               IF NOT "IX_MPO_RefSwitchOvenFeederOutside_I7" AND "IX_MPO_RefSwitchOvenFeederInside_I6"
                   AND "IX_MPO_RefSwitchVac_PosTurnTable_I5" AND NOT "IX_MPO_RefSwitchVac_PosOven_I8" THEN
                   "QX_MPO_M5_VacuumTowardsOven_Q7" := FALSE;
                   "QX_MPO_M5_VacuumTowardsTurnTable_Q8" := FALSE;
                   "QX_MPO_M4_OvenFeederRetract_Q5" := FALSE;
                   "QX_MPO_M4_OvenFeederExtend_Q6" := FALSE;
                   "QX_MPO_ValveOvenDoor_Q13" := FALSE;
                   #li_StepCase := 200;
               END_IF;

           200: // vacuum suction device down at turn table
               IF "IX_MPO_RefSwitchTurnTable_PosVac_I1" THEN
                   "QX_MPO_ValveLowering_Q12" := TRUE;

                   #lx_Start_TON_Wait := TRUE;
                   #lt_TON_Wait := T#2000ms;

                   IF #lfb_TON_Wait.Q THEN
                       #lx_Start_TON_Wait := FALSE;
                       #li_StepCase := 210;
                   END_IF;
               END_IF;

           210: // vacuum off
               "QX_MPO_ValveVacuum_Q11" := FALSE;

               #lx_Start_TON_Wait := TRUE;
               #lt_TON_Wait := T#2000ms;

               IF #lfb_TON_Wait.Q THEN
                   #lx_Start_TON_Wait := FALSE;
                   #li_StepCase := 220;
               END_IF;

           220: // vacuum suction device up
               "QX_MPO_ValveLowering_Q12" := FALSE;

               #lx_Start_TON_Wait := TRUE;
               #lt_TON_Wait := T#2000ms;

               IF #lfb_TON_Wait.Q THEN
                   #lx_Start_TON_Wait := FALSE;
                   IF "gtyp_MPO".Workpiece_Parameters.DoSaw THEN
                       #li_StepCase := 230;
                   ELSE    //Just skip the saw all together
                       #li_StepCase := 251;
                   END_IF;
               END_IF;

           230: // Position turn table saw
               IF NOT "IX_MPO_RefSwitchTurnTable_PosSaw_I4" AND NOT "IX_MPO_RefSwitchTurnTable_PosBelt_I2" AND "IX_MPO_RefSwitchTurnTable_PosVac_I1" THEN
                   "QX_MPO_M1_TurnTableClockwise_Q1" := TRUE;
                   "QX_MPO_M1_TurnTableCounterclockwise_Q2" := FALSE;
               ELSIF "IX_MPO_RefSwitchTurnTable_PosSaw_I4" OR "IX_MPO_RefSwitchTurnTable_PosBelt_I2" AND NOT "IX_MPO_RefSwitchTurnTable_PosVac_I1" THEN
                   "QX_MPO_M1_TurnTableClockwise_Q1" := FALSE;
                   "QX_MPO_M1_TurnTableCounterclockwise_Q2" := FALSE;

                   // Update workpiece state to saw on and update timestamp
                   "gtyp_MPO".Workpiece.Workpiece_States.x_atSaw := TRUE;
                   "gtyp_MPO".Workpiece.Workpiece_States.ldt_Saw := DT_TO_LDT(#ldt_MQTT);

                   #li_StepCase := 240;
               END_IF;

           240: // Start sawing
               "QX_MPO_M3_Saw_Q4" := TRUE;



               #lx_Start_TON_Wait := TRUE;
               #lt_TON_Wait := "gtyp_MPO".Workpiece_Parameters.SawTime; //Replaced the default sawing time of T#4000ms with the variable

               IF #lfb_TON_Wait.Q THEN
                   #li_Return_LDT := RD_SYS_T(#ldt_MQTT);
                   "gtyp_MPO".History[6].i_code := 600;
                   "gtyp_MPO".History[6].ldt_ts := DT_TO_LDT(#ldt_MQTT);

                   #lx_Start_TON_Wait := FALSE;

                   //TURN OFF SAW
                   "QX_MPO_M3_Saw_Q4" := FALSE;

                   // Update workpiece state to saw off and update timestamp
                   "gtyp_MPO".Workpiece.Workpiece_States.x_atSaw := FALSE;
                   "gtyp_MPO".Workpiece.Workpiece_States.ldt_Saw := DT_TO_LDT(#ldt_MQTT);

                   #li_StepCase := 250;
               END_IF;

           250: // Position turn table Pos Belt
               IF "IX_MPO_RefSwitchTurnTable_PosSaw_I4" AND NOT "IX_MPO_RefSwitchTurnTable_PosBelt_I2" AND NOT "IX_MPO_RefSwitchTurnTable_PosVac_I1" THEN
                   "QX_MPO_M1_TurnTableClockwise_Q1" := TRUE;
                   "QX_MPO_M1_TurnTableCounterclockwise_Q2" := FALSE;
               ELSIF NOT "IX_MPO_RefSwitchTurnTable_PosSaw_I4" AND "IX_MPO_RefSwitchTurnTable_PosBelt_I2" AND NOT "IX_MPO_RefSwitchTurnTable_PosVac_I1" THEN
                   "QX_MPO_M1_TurnTableClockwise_Q1" := FALSE;
                   "QX_MPO_M1_TurnTableCounterclockwise_Q2" := FALSE;
                   #li_StepCase := 260;
               END_IF;

           251: // Position turn table Pos Belt Directly (this has been added by me)
               IF NOT "IX_MPO_RefSwitchTurnTable_PosBelt_I2" THEN
                   "gtyp_MPO"."i_PWM_TurnTable" := 700;
                   "QX_MPO_M1_TurnTableClockwise_Q1" := TRUE;
                   "QX_MPO_M1_TurnTableCounterclockwise_Q2" := FALSE;
               ELSIF NOT "IX_MPO_RefSwitchTurnTable_PosSaw_I4" AND "IX_MPO_RefSwitchTurnTable_PosBelt_I2" AND NOT "IX_MPO_RefSwitchTurnTable_PosVac_I1" THEN
                   "gtyp_MPO"."i_PWM_TurnTable" := 1000;
                   "QX_MPO_M1_TurnTableClockwise_Q1" := FALSE;
                   "QX_MPO_M1_TurnTableCounterclockwise_Q2" := FALSE;
                   #li_StepCase := 260;
               END_IF;

           260: // put workpiece to belt
               "QX_MPO_ValveFeeder_Q14" := TRUE;

               #lx_Start_TON_Wait := TRUE;
               #lt_TON_Wait := T#1000ms;

               IF #lfb_TON_Wait.Q THEN
                   #lx_Start_TON_Wait := FALSE;
                   "QX_MPO_ValveFeeder_Q14" := FALSE;
                   "QX_MPO_Compressor_Q10" := FALSE;
                   #li_StepCase := 270;
               END_IF;

           270: // Position turn table Pos Vacuum
               IF "IX_MPO_RefSwitchTurnTable_PosSaw_I4" OR "IX_MPO_RefSwitchTurnTable_PosBelt_I2" OR NOT "IX_MPO_RefSwitchTurnTable_PosVac_I1" THEN
                   "QX_MPO_M1_TurnTableClockwise_Q1" := FALSE;
                   "QX_MPO_M1_TurnTableCounterclockwise_Q2" := TRUE;
               ELSIF NOT "IX_MPO_RefSwitchTurnTable_PosSaw_I4" AND NOT "IX_MPO_RefSwitchTurnTable_PosBelt_I2" AND "IX_MPO_RefSwitchTurnTable_PosVac_I1" THEN
                   "QX_MPO_M1_TurnTableClockwise_Q1" := FALSE;
                   "QX_MPO_M1_TurnTableCounterclockwise_Q2" := FALSE;
                   "QX_MPO_Compressor_Q10" := FALSE;
                   #li_StepCase := 280;
               END_IF;

           280: // Start conveyor belt
               "QX_MPO_M2_ConveyorBeltForward_Q3" := TRUE;

               #lx_Time_Error := TRUE;

               IF #lfb_TOF_ConveyerBelt_Out.Q THEN
                   "gtyp_SLD".History := "gtyp_MPO".History;
                   "gtyp_SLD".Workpiece := "gtyp_MPO".Workpiece;
                   "gtyp_MPO".Workpiece.s_id := '0';
                   "gtyp_MPO".Workpiece.s_state := '';
                   "gtyp_MPO".Workpiece.s_type := '';
                   FOR #ti_Counter := 1 TO 8 DO
                       "gtyp_MPO".History[#ti_Counter].i_code := 0;
                       "gtyp_MPO".History[#ti_Counter].ldt_ts := DT#1990-01-01-00:00:00;
                   END_FOR;

                   "gtyp_Interface_Dashboard".Subscribe.State_MPO.x_active := FALSE;

                   #lx_Time_Error := FALSE;
                   #li_StepCase := 290;
               END_IF;

               // runtime error
               IF #lfb_TON_Error.Q THEN
                   #li_Lights := 4;
                   #lx_Time_Error := FALSE;
                   "QX_MPO_M2_ConveyorBeltForward_Q3" := FALSE;
                   "gtyp_Interface_Dashboard".Subscribe.State_MPO.x_active := FALSE;
                   "gtyp_MPO".x_Error := TRUE;
                   "gtyp_MPO".s_ErrorMessage := 'MPO RUNTIME ERROR';
                   #li_StepCase := 0;
               END_IF;

           290: // wait for runtime on conveyor belt

               IF NOT #lfb_TOF_ConveyerBelt_Out.Q THEN
                   #lx_Start_TON_Wait := FALSE;
                   "QX_MPO_M2_ConveyorBeltForward_Q3" := FALSE;
                   #li_StepCase := 60;
               END_IF;
               // Statement section ELSE
           ELSE
               ;
       END_CASE;

       "QW_MPO_PWM_TurnTable_M1" := "gtyp_MPO"."i_PWM_TurnTable";
       "QW_MPO_PWM_Vacuum_M5" := "gtyp_MPO"."i_PWM_Vacuum";

   ELSE
       #li_Lights := 1;
       #lx_Init := TRUE;
       "gtyp_MPO".x_Start_Park_Position := FALSE;
       "gtyp_MPO".x_Park_Position_Reached := FALSE;
   END_IF;
END_FUNCTION_BLOCK

FUNCTION_BLOCK "PRG_MPO_Set_Park_Position"   // FB39, SCL
TITLE = Program Set Positioning HBW
{ S7_Optimized_Access := 'TRUE' }
AUTHOR : A.Schaefer
VERSION : 0.0
   VAR
      lx_Init : Bool;
      lx_Start_TON_Wait : Bool;
      lt_TON_Wait : Time;
      li_StepCase : Int;
      lfb_TON_Wait : TON_TIME;
      lfb_R_Trig_Start_Park_Pos : R_TRIG;
   END_VAR
BEGIN
   IF #lx_Init THEN

       // FB TON Wait
       #lfb_TON_Wait(IN := #lx_Start_TON_Wait,
                     PT := #lt_TON_Wait);

       #lfb_R_Trig_Start_Park_Pos(CLK := "gtyp_Setup".x_Park_Position
                                  OR "IX_Set_Park_Position");

       // Set Start Park Position   
       IF #lfb_R_Trig_Start_Park_Pos.Q THEN
           "gtyp_MPO".x_Start_Park_Position := TRUE;
           #li_StepCase := 0;
       END_IF;

       // not Start Park Pos Step 0
       IF NOT "gtyp_MPO".x_Start_Park_Position THEN
           #li_StepCase := 0;
       END_IF;

       // step chain HBW
       CASE #li_StepCase OF

           0:  // init
               #lx_Start_TON_Wait := FALSE;
               #li_StepCase := 10;

           10:  // Set Positioning activ?
               IF "gtyp_MPO".x_Start_Park_Position AND NOT "gtyp_MPO".x_Park_Position_Reached THEN
                   #li_StepCase := 20;
               END_IF;

           20: // Towards
               "QX_MPO_M5_VacuumTowardsTurnTable_Q8" := FALSE;
               "QX_MPO_M5_VacuumTowardsOven_Q7" := TRUE;
               #lx_Start_TON_Wait := TRUE;
               #lt_TON_Wait := T#4000ms;

               IF #lfb_TON_Wait.Q THEN
                   "QX_MPO_M5_VacuumTowardsTurnTable_Q8" := FALSE;
                   "QX_MPO_M5_VacuumTowardsOven_Q7" := FALSE;
                   #lx_Start_TON_Wait := FALSE;
                   #li_StepCase := 30;
               END_IF;

           30: // homing vertical axis
               "QX_MPO_M1_TurnTableClockwise_Q1" := TRUE;
               "QX_MPO_M1_TurnTableCounterclockwise_Q2" := FALSE;
               #lx_Start_TON_Wait := TRUE;
               #lt_TON_Wait := T#1000ms;

               IF #lfb_TON_Wait.Q THEN
                   "QX_MPO_M1_TurnTableClockwise_Q1" := FALSE;
                   "QX_MPO_M1_TurnTableCounterclockwise_Q2" := FALSE;
                   #lx_Start_TON_Wait := FALSE;
                   #li_StepCase := 40;
               END_IF;

           40: // Deciding which doing
               "gtyp_MPO".x_Park_Position_Reached := TRUE;


               // Statement section ELSE    
           ELSE
               ;
       END_CASE;

   ELSE
       #lx_Init := TRUE;
   END_IF;
END_FUNCTION_BLOCK

// folder: NFC

FUNCTION_BLOCK "PRG_NFC"   // FB8, SCL
TITLE = Program NFC
{ S7_Optimized_Access := 'TRUE' }
AUTHOR : A.Schaefer
VERSION : 0.0
   VAR
      lx_Init : Bool;
      lx_Start : Bool;
      lx_Time_Wait : Bool;
      lx_Time_Error : Bool;
      li_StepCase : Int;
      ldt_MQTT : Date_And_Time;
      ldt_Delete_old : LDT;
      ldt_Read_old : LDT;
      li_Return_LDT : Int;
      lfb_TON_Error : TON_TIME;
      lfb_TON_Wait : TON_TIME;
   END_VAR
BEGIN
   IF #lx_Init THEN

       // runtime monitoring error
       #lfb_TON_Error(IN := #lx_Time_Error,
                      PT := T#30s);

       // runtime monitoring read uid
       #lfb_TON_Wait(IN := #lx_Time_Wait,
                     PT := T#5s);

       // step chain NFC
       CASE #li_StepCase OF

           0:  // init
               #lx_Time_Wait := FALSE;
               "gtyp_VGR"."x_NFC_Completed" := FALSE;

               // delete and write first state to chip
               IF "gtyp_VGR".x_NFC_Start_First AND NOT "gtyp_VGR".x_Workpiece_NiO THEN
                   "gtyp_Interface_TXT_Controler".Subscribe.State_NFC_Device.Workpiece.s_state := '';
                   "gtyp_Interface_TXT_Controler".Subscribe.State_NFC_Device.Workpiece.s_type := '';

                   "gtyp_Interface_TXT_Controler".Publish.ActionButtonNFCModule.s_cmd := '';
                   #li_StepCase := 10;
                   // write color or processed finished to chip
               ELSIF "gtyp_VGR".x_NFC_Start AND NOT "gtyp_VGR".x_Workpiece_NiO THEN
                   "gtyp_Interface_TXT_Controler".Publish.ActionButtonNFCModule.s_cmd := '';
                   #li_StepCase := 40;
                   // read chip for delete HBW
               ELSIF "QX_SSC_LED_Green_Q5" AND NOT "gtyp_VGR".x_Workpiece_NiO THEN
                   #ldt_Read_old := "gtyp_Interface_Dashboard".Publish.ActionButtonNFCModule.ldt_ts;
                   "gtyp_VGR".x_NFC_Start_First := FALSE;
                   "gtyp_VGR".x_NFC_Start := FALSE;
                   "gtyp_Interface_TXT_Controler".Publish.ActionButtonNFCModule.s_cmd := '';
                   #li_StepCase := 60;
               END_IF;

           10: // delete

               "gtyp_Interface_TXT_Controler".Publish.ActionButtonNFCModule.s_cmd := 'delete';
               #li_Return_LDT := RD_SYS_T(#ldt_MQTT);
               "gtyp_Interface_TXT_Controler".Publish.ActionButtonNFCModule.ldt_ts := DT_TO_LDT(#ldt_MQTT);

               #li_StepCase := 20;

           20: // wait to answer from dashboard
               #lx_Time_Error := TRUE;
               IF ("gtyp_Interface_TXT_Controler".Subscribe.State_NFC_Device.ldt_ts > "gtyp_Interface_TXT_Controler".Publish.ActionButtonNFCModule.ldt_ts)
                   AND ("gtyp_Interface_TXT_Controler".Subscribe.State_NFC_Device.Workpiece.s_type = 'NONE')
                   AND ("gtyp_Interface_TXT_Controler".Subscribe.State_NFC_Device.Workpiece.s_state <> '')
                   AND ("gtyp_Interface_TXT_Controler".Subscribe.State_NFC_Device.Workpiece.s_id <> '') THEN
                   "gtyp_VGR".Workpiece.s_id := "gtyp_Interface_TXT_Controler".Subscribe.State_NFC_Device.Workpiece.s_id;
                   #lx_Time_Error := FALSE;
                   #li_StepCase := 30;
               END_IF;
               // runtime error
               IF #lfb_TON_Error.Q THEN
                   #lx_Time_Error := FALSE;
                   "gtyp_VGR".x_Workpiece_NiO := TRUE;
                   #li_StepCase := 0;
               END_IF;


           30: // wait of answer 
               IF "gtyp_Interface_TXT_Controler".Subscribe.State_NFC_Device.Workpiece.s_id <> '' THEN
                   #li_StepCase := 40;
               END_IF;

           40:  // write
               "gtyp_Interface_TXT_Controler".Publish.ActionButtonNFCModule.History := "gtyp_VGR".History;
               "gtyp_Interface_TXT_Controler".Publish.ActionButtonNFCModule.Workpiece.s_type := "gtyp_VGR".Workpiece.s_type;
               "gtyp_Interface_TXT_Controler".Publish.ActionButtonNFCModule.Workpiece.s_state := "gtyp_VGR".Workpiece.s_state;

               #li_Return_LDT := RD_SYS_T(#ldt_MQTT);

               "gtyp_Interface_TXT_Controler".Publish.ActionButtonNFCModule.s_cmd := 'write';
               "gtyp_Interface_TXT_Controler".Publish.ActionButtonNFCModule.ldt_ts := DT_TO_LDT(#ldt_MQTT);

               #li_StepCase := 50;

           50: // wait of answer write 
               #lx_Time_Error := TRUE;
               IF ("gtyp_Interface_TXT_Controler".Subscribe.State_NFC_Device.ldt_ts > "gtyp_Interface_TXT_Controler".Publish.ActionButtonNFCModule.ldt_ts) THEN
                   #lx_Time_Error := FALSE;
                   #li_StepCase := 80;
               END_IF;
               // runtime error
               IF #lfb_TON_Error.Q THEN
                   #lx_Time_Error := FALSE;
                   "gtyp_VGR".x_Workpiece_NiO := TRUE;
                   #li_StepCase := 0;
               END_IF;

           60: // read uid cmd

               #li_Return_LDT := RD_SYS_T(#ldt_MQTT);

               "gtyp_Interface_TXT_Controler".Publish.ActionButtonNFCModule.s_cmd := 'read_uid';
               "gtyp_Interface_TXT_Controler".Publish.ActionButtonNFCModule.ldt_ts := DT_TO_LDT(#ldt_MQTT);
               #lx_Time_Wait := TRUE;
               #li_StepCase := 70;

           70: // wait of answer read_uid 
               IF NOT "QX_SSC_LED_Green_Q5" OR #lfb_TON_Wait.Q OR ("gtyp_Interface_TXT_Controler".Subscribe.State_NFC_Device.ldt_ts > "gtyp_Interface_TXT_Controler".Publish.ActionButtonNFCModule.ldt_ts) THEN
                   IF LEN("gtyp_Interface_TXT_Controler".Subscribe.State_NFC_Device.Workpiece.s_id) = 8 THEN
                       "gtyp_Setup".x_Clean_Rack_HBW := TRUE;
                   END_IF;
                   #lx_Time_Wait := FALSE;
                   "gtyp_Interface_TXT_Controler".Subscribe.State_NFC_Device.Workpiece.s_id := '';
                   #li_StepCase := 0;
               END_IF;

           80: // completed

               "gtyp_VGR"."x_NFC_Completed" := TRUE;

               IF NOT "gtyp_VGR".x_NFC_Start AND NOT "gtyp_VGR".x_NFC_Start_First THEN
                   "gtyp_VGR"."x_NFC_Completed" := FALSE;
                   #lx_Start := FALSE;
                   #li_StepCase := 0;
               END_IF;

               // Statement section ELSE
           ELSE
               ;
       END_CASE;

   ELSE
       #lx_Init := TRUE;
   END_IF;
END_FUNCTION_BLOCK

// folder: Order

FUNCTION_BLOCK "PRG_Order"   // FB20, SCL
TITLE = Program Order
{ S7_Optimized_Access := 'TRUE' }
AUTHOR : A.Schaefer
VERSION : 0.0
   VAR
      lx_Init : Bool;
      li_StepCase : Int;
      lldt_ts_old : LDT;
      ldt_MQTT : Date_And_Time;
      li_Return_LDT : Int;
      lfb_TON_Wait : TON_TIME;
      lx_Start_TON_Wait : Bool;
   END_VAR
   VAR_TEMP
      ti_Que_Counter : Int;
      ti_Que_Output : Int;
   END_VAR
BEGIN
   IF #lx_Init THEN
       #lfb_TON_Wait(IN := #lx_Start_TON_Wait,
                     PT := T#20s);

       // step chain order
       CASE #li_StepCase OF

           0:  // init
               #lx_Start_TON_Wait := FALSE;
               #li_StepCase := 10;

           10: // check whether order button has been pressed (time stamp changes)

               IF ("gtyp_Interface_Dashboard".Publish.OrderWorkpieceButton.ldt_ts > #lldt_ts_old) THEN
                   #lldt_ts_old := "gtyp_Interface_Dashboard".Publish.OrderWorkpieceButton.ldt_ts;
                   IF ("Queue".i_Queue_Index < "Ci_Queue_Length") THEN
                       "Queue".Queue["Queue".i_Queue_Index] := "gtyp_Interface_Dashboard".Publish.OrderWorkpieceButton;
                       #li_Return_LDT := RD_SYS_T(#ldt_MQTT);
                       "gtyp_Interface_Dashboard".Subscribe.State_Order.ldt_ts := DT_TO_LDT(#ldt_MQTT);
                       "gtyp_Interface_Dashboard".Subscribe.State_Order.s_state := 'ORDERED';
                       "gtyp_Interface_Dashboard".Subscribe.State_Order.s_type := "Queue".Queue["Queue".i_Queue_Index].s_type;
                       "Queue".i_Queue_Index += 1;
                       IF ("Queue".i_Queue_Index = "Ci_Queue_Length") THEN
                           "Queue".x_Queue_Full := TRUE;
                       END_IF;
                   END_IF;
                   //Reset the parameters when the order has been processed
                   "gtyp_Interface_Dashboard".Publish.OrderWorkpieceButton.Workpiece_Parameters := "Queue".Queue["Ci_Queue_Length"].Workpiece_Parameters;
               END_IF;

               //There is an order in the que
               IF ("Queue".i_Queue_Index > 0) THEN
                   //The VGR is ready to start with the next product in the que
                   IF "gtyp_VGR".x_Ready_For_Order AND "gtyp_VGR".x_Ready_For_Outsource THEN
                       //We want to output the first order
                       FOR #ti_Que_Output := 0 TO "Queue".i_Queue_Index - 1 DO
                           IF ("Queue".Queue[#ti_Que_Output].s_type = 'RED' AND "gtyp_HBW".i_Red_Available = 0) THEN
                               CONTINUE;
                           ELSIF ("Queue".Queue[#ti_Que_Output].s_type = 'BLUE' AND "gtyp_HBW".i_Blue_Available = 0) THEN
                               CONTINUE;
                           ELSIF ("Queue".Queue[#ti_Que_Output].s_type = 'WHITE' AND "gtyp_HBW".i_White_Available = 0) THEN
                               CONTINUE;
                           END_IF;
                           //Possible order found
                           //Set index back
                           "Queue".i_Queue_Index -= 1;
                           "Queue".x_Queue_Full := FALSE;
                           //VGR is ready
                           "gtyp_VGR".x_Ready_For_Order := FALSE;
                           //Copy que to VGR
                           "gtyp_VGR".s_HBW_Outsource_Typ := "Queue".Queue[#ti_Que_Output].s_type;
                           "gtyp_VGR".Worpiece_Parameters := "Queue".Queue[#ti_Que_Output].Workpiece_Parameters;

                           //ADDED TO MAKE DISPLAYING PARAMETERS ON DASHBOARD EASIER
                           "gtyp_VGR".Workpiece.Workpiece_Parameters := "Queue".Queue[#ti_Que_Output].Workpiece_Parameters;
                           //Shift que
                           FOR #ti_Que_Counter := #ti_Que_Output TO "Ci_Queue_Length" - 1 DO
                               "Queue".Queue[#ti_Que_Counter] := "Queue".Queue[#ti_Que_Counter + 1];
                           END_FOR;
                           //Start the HBW and VGR
                           "gtyp_VGR".x_HBW_Outsource := TRUE;
                           EXIT;
                       END_FOR;
                   END_IF;
               END_IF;

               IF "gtyp_VGR".x_HBW_PickedUp THEN
                   "gtyp_VGR".x_HBW_Outsource := FALSE;
                   "gtyp_VGR".s_HBW_Outsource_Typ := '';
                   #li_StepCase := 0;
               END_IF;

               // Statement section ELSE
           ELSE
               ;
       END_CASE;

   ELSE
       #lx_Init := TRUE;
       "Queue".i_Queue_Index := 0;
       "Queue".x_Queue_Full := FALSE;
       #lldt_ts_old := LDT#1970-01-01-00:00:00;
   END_IF;
END_FUNCTION_BLOCK

// folder: SLD_Sorting_Line_With_Color_Detection

FUNCTION_BLOCK "PRG_SLD_Calibration_Color"   // FB33, SCL
TITLE = Program Calibration Color Sensor SLD
{ S7_Optimized_Access := 'TRUE' }
AUTHOR : A.Schaefer
VERSION : 0.0
   VAR
      lx_Init : Bool;
      lx_Start_TON_Wait : Bool;
      lx_Start_Positioning_m : Bool;
      lt_TON_Wait : Time;
      li_StepCase : Int;
      lw_ColorValueMin : Word;
      ldi_Pos_Horizontal : DInt;
      ldi_Pos_Vertical : DInt;
      lfb_R_Trig_Deaktivate : R_TRIG;
      lfb_TON_Wait : TON_TIME;
   END_VAR
BEGIN
   IF #lx_Init THEN

       // FB TON Wait
       #lfb_TON_Wait(IN := #lx_Start_TON_Wait,
                     PT := #lt_TON_Wait);

       #lfb_R_Trig_Deaktivate(CLK := NOT "gtyp_Setup".x_Color_Sensor_Calibration
                              OR NOT ("gtyp_Setup".i_Color_Sensor_Selection = 2));
       // Deaktivate step 0   
       IF #lfb_R_Trig_Deaktivate.Q THEN
           "gtyp_Setup".x_Calculate_Value_Color := FALSE;
           "gtyp_Setup".x_Set_Calib_Value_Color_Blue := FALSE;
           "gtyp_Setup".x_Set_Calib_Value_Color_Red := FALSE;
           "gtyp_Setup".x_Set_Calib_Value_Color_White := FALSE;
           "gtyp_Setup".w_Calib_ColorValue_Blue := 0;
           "gtyp_Setup".w_Calib_ColorValue_Red := 0;
           "gtyp_Setup".w_Calib_ColorValue_White := 0;
           "gtyp_Setup".w_Threshold_Red_Blue := 0;
           "gtyp_Setup".w_Threshold_White_Red := 0;
           "QX_SLD_M1_ConveyorBelt_Q1" := FALSE;
           #lw_ColorValueMin := 16#FF;
           #li_StepCase := 0;
       END_IF;

       // step chain HBW
       CASE #li_StepCase OF

           0:  // init
               #lx_Start_TON_Wait := FALSE;
               #li_StepCase := 10;

           10:  // Set Calibration activ?
               IF "gtyp_Setup".x_Color_Sensor_Calibration
                   AND ("gtyp_Setup".i_Color_Sensor_Selection = 2) THEN
                   "gtyp_Setup".x_Calculate_Value_Color := FALSE;
                   "gtyp_Setup".x_Set_Calib_Value_Color_Blue := FALSE;
                   "gtyp_Setup".x_Set_Calib_Value_Color_Red := FALSE;
                   "gtyp_Setup".x_Set_Calib_Value_Color_White := FALSE;
                   "gtyp_Setup".w_Calib_ColorValue_Blue := 0;
                   "gtyp_Setup".w_Calib_ColorValue_Red := 0;
                   "gtyp_Setup".w_Calib_ColorValue_White := 0;
                   "gtyp_Setup".w_Threshold_Red_Blue := 0;
                   "gtyp_Setup".w_Threshold_White_Red := 0;
                   "QX_SLD_M1_ConveyorBelt_Q1" := FALSE;
                   #lw_ColorValueMin := 16#FFFF;
                   #li_StepCase := 20;
               END_IF;

           20: // wait for set Values or Calculate

               IF NOT "IX_SLD_LightBarrierInlet_I2" THEN
                   "QX_SLD_M1_ConveyorBelt_Q1" := TRUE;
                   #lw_ColorValueMin := 16#FFFF;
               END_IF;

               IF #lw_ColorValueMin > "IW_SLD_ColorSensor_A4" THEN
                   #lw_ColorValueMin := "IW_SLD_ColorSensor_A4";
               END_IF;

               IF NOT "IX_SLD_LightBarrierBehindColorSensor_I3" THEN
                   "QX_SLD_M1_ConveyorBelt_Q1" := FALSE;
               END_IF;

               // Start new Positioning
               IF "gtyp_Setup".x_Set_Calib_Value_Color_Blue THEN
                   "gtyp_Setup".w_Calib_ColorValue_Blue := #lw_ColorValueMin;
                   "gtyp_Setup".x_Set_Calib_Value_Color_Blue := FALSE;
               ELSIF "gtyp_Setup".x_Set_Calib_Value_Color_Red THEN
                   "gtyp_Setup".w_Calib_ColorValue_Red := #lw_ColorValueMin;
                   "gtyp_Setup".x_Set_Calib_Value_Color_Red := FALSE;
               ELSIF "gtyp_Setup".x_Set_Calib_Value_Color_White THEN
                   "gtyp_Setup".w_Calib_ColorValue_White := #lw_ColorValueMin;
                   "gtyp_Setup".x_Set_Calib_Value_Color_White := FALSE;
               END_IF;

               "gtyp_Setup".w_Threshold_White_Red := "gtyp_Setup".w_Calib_ColorValue_White + (("gtyp_Setup".w_Calib_ColorValue_Red - "gtyp_Setup".w_Calib_ColorValue_White) / 2);
               "gtyp_Setup".w_Threshold_Red_Blue := "gtyp_Setup".w_Calib_ColorValue_Red + (("gtyp_Setup".w_Calib_ColorValue_Blue - "gtyp_Setup".w_Calib_ColorValue_Red) / 2);

               IF "gtyp_Setup".x_Calculate_Value_Color THEN
                   "gtyp_SLD".w_Threshold_White_Red := "gtyp_Setup".w_Threshold_White_Red;
                   "gtyp_SLD".w_Threshold_Red_Blue := "gtyp_Setup".w_Threshold_Red_Blue;
                   "gtyp_Setup".x_Calculate_Value_Color := FALSE;
               END_IF;

               // Statement section ELSE    
           ELSE
               ;
       END_CASE;

       IF ("gtyp_Setup".i_Color_Sensor_Selection = 2) THEN
           // Reload Pos Value
           "gtyp_Setup".w_Actual_ColorValue := "IW_SLD_ColorSensor_A4";
       END_IF;
   ELSE
       #lx_Init := TRUE;
   END_IF;
END_FUNCTION_BLOCK

FUNCTION_BLOCK "PRG_SLD_Set_Counter_Values"   // FB34, SCL
TITLE = Program Set counter Values SLD
{ S7_Optimized_Access := 'TRUE' }
AUTHOR : A.Schaefer
VERSION : 0.0
   VAR
      lx_Init : Bool;
      lfb_R_Trig_Calib_activ : R_TRIG;
   END_VAR
BEGIN
   IF #lx_Init THEN

       // Reload act. Counter Values
       IF NOT "gtyp_Setup".x_Counter_Value_Calibration THEN
           "gtyp_Setup".i_Calib_CounterValue_Blue := "gtyp_SLD".i_CounterValue_Blue;
           "gtyp_Setup".i_Calib_CounterValue_Red := "gtyp_SLD".i_CounterValue_Red;
           "gtyp_Setup".i_Calib_CounterValue_White := "gtyp_SLD".i_CounterValue_White;
       END_IF;

       // Set Counter Values   
       IF "gtyp_Setup".x_Set_CounterValues AND "gtyp_Setup".x_Counter_Value_Calibration THEN
           "gtyp_SLD".i_CounterValue_Blue := "gtyp_Setup".i_Calib_CounterValue_Blue;
           "gtyp_SLD".i_CounterValue_Red := "gtyp_Setup".i_Calib_CounterValue_Red;
           "gtyp_SLD".i_CounterValue_White := "gtyp_Setup".i_Calib_CounterValue_White;
           "gtyp_Setup".x_Set_CounterValues := FALSE;
       END_IF;

   ELSE
       #lx_Init := TRUE;
   END_IF;
END_FUNCTION_BLOCK

// folder: SSC_Sensor_Station_With_Camera

FUNCTION_BLOCK "PRG_SSC_Axis_Vertical"   // FB11, SCL
TITLE = Program Axis vertical SSC
{ S7_Optimized_Access := 'TRUE' }
AUTHOR : A.Schaefer
VERSION : 0.0
   VAR
      lx_Init : Bool;
      lfb_Vertical_Axis : "FB_Axis";
   END_VAR
BEGIN
   IF #lx_Init THEN

       // FB Axis vertical
       #lfb_Vertical_Axis(ini_Axis := 5,
                          indi_Increment := "gtyp_SSC".Vertical_Axis.di_Increment,
                          inx_Ref_Switch := "IX_SSC_RefSwitchVerticalAxis_I1",
                          inx_Referencing := "gtyp_SSC".Vertical_Axis.x_Reference,
                          inx_Start_Positioning := "gtyp_SSC".Vertical_Axis.x_Start_Positioning,
                          indi_Target_Position := "gtyp_SSC".Vertical_Axis.di_Target_Position,
                          ini_PWM := "gtyp_SSC".Vertical_Axis.i_PWM,
                          inouttyp_Config := "gtyp_SSC".Vertical_Axis.Config,
                          inouttyp_Setup := "gtyp_SetupAxis");

       "QX_SSC_M1_VerticalAxisUp_Q1" := #lfb_Vertical_Axis.outx_Motor_Pos;
       "QX_SSC_M1_VerticalAxisDown_Q2" := #lfb_Vertical_Axis.outx_Motor_Neg;
       "QW_SSC_PWM_Vertical_M1" := #lfb_Vertical_Axis.outi_Motor_PWM;
       "gtyp_SSC".Vertical_Axis.di_Actual_Position := #lfb_Vertical_Axis.outdi_Actual_Position;
       "gtyp_SSC".Vertical_Axis.x_Referenced := #lfb_Vertical_Axis.outx_Referenced;
       "gtyp_SSC".Vertical_Axis.x_Position_Reached := #lfb_Vertical_Axis.outx_Position_Reached;
   ELSE
       #lx_Init := TRUE;
   END_IF;
END_FUNCTION_BLOCK

FUNCTION_BLOCK "PRG_SSC_Ablauf"   // FB12, SCL
TITLE = Program Ablauf SSC
{ S7_Optimized_Access := 'TRUE' }
AUTHOR : A.Schaefer
VERSION : 0.0
   VAR
      lx_Init : Bool;
      lx_FirstCentre : Bool;
      lx_Start : Bool;
      lx_Start_TON_State : Bool;
      lt_TON_Wait : Time;
      li_StepCase : Int;
      ldi_TargetPosition_Horizontal : DInt;
      ldi_TargetPosition_Vertical : DInt;
      lldt_ts_old : LDT;
      ldt_write : Date_And_Time;
      li_Return_write : Int;
      ldt_MQTT : Date_And_Time;
      li_Return_LDT : Int;
      lx_Start_TON_Wait : Bool;
      ldi_StepHorizontal : DInt;
      ldi_StepVertical : DInt;
      lfb_TON_Wait : TON_TIME;
      lfb_TON_State : TON_TIME;
      lfb_F_TRIG_Set_Pos : F_TRIG;
   END_VAR
BEGIN
   IF #lx_Init THEN

       // Restart after set Positioning
       IF "gtyp_Setup".x_Set_Pos_Activ OR "gtyp_SSC".x_Start_Park_Position THEN
           #li_StepCase := 0;
       END_IF;

       // falling edge Set Pos
       #lfb_F_TRIG_Set_Pos(CLK := "gtyp_Setup".x_Set_Pos_Activ);

       IF #lfb_F_TRIG_Set_Pos.Q THEN
           #lx_FirstCentre := TRUE;
       END_IF;

       #lfb_TON_Wait(IN := #lx_Start_TON_Wait,
                     PT := #lt_TON_Wait);

       // wait time state
       #lfb_TON_State(IN := NOT #lx_Start_TON_State,
                      PT := T#2s);

       // state of the ssc cyclically transmitted to the cloud
       IF #lfb_TON_State.Q AND NOT #lx_Start_TON_State THEN
           #lx_Start_TON_State := TRUE;
           #li_Return_LDT := RD_SYS_T(#ldt_MQTT);
           "gtyp_Interface_Dashboard".Subscribe.PosPanTiltUnit.ldt_ts := DT_TO_LDT(#ldt_MQTT);
       END_IF;

       // restart wait time state
       IF NOT #lfb_TON_State.Q AND #lx_Start_TON_State THEN
           #lx_Start_TON_State := FALSE;
       END_IF;

       CASE #li_StepCase OF

           0:  // Init
               #lx_Start_TON_State := FALSE;
               "gtyp_SSC".Horizontal_Axis.x_Start_Positioning := FALSE;
               "gtyp_SSC".Vertical_Axis.x_Start_Positioning := FALSE;

               IF NOT "gtyp_Setup".x_Set_Pos_Activ AND NOT "gtyp_SSC".x_Start_Park_Position THEN
                   #li_StepCase := 10;
               END_IF;

           10: // Deciding which route to take 

               IF ("gtyp_Interface_Dashboard".Publish.PosPanTiltUnit.ldt_ts > #lldt_ts_old) OR #lx_FirstCentre THEN

                   #lldt_ts_old := "gtyp_Interface_Dashboard".Publish.PosPanTiltUnit.ldt_ts;

                   // convert the degrees to position
                   #ldi_StepHorizontal := REAL_TO_DINT("FC_Scale_linear"(inr_Y1 := DINT_TO_REAL("gtyp_SSC".Horizontal_Axis.Config.di_Neg_Soft_Switch),
                                                                                                             inr_Y2 := DINT_TO_REAL("gtyp_SSC".Horizontal_Axis.Config.di_Pos_Soft_Switch),
                                                                                                             inr_X1 := 0.0,
                                                                                                             inr_X2 := 180.0,
                                                                                                             inr_X := DINT_TO_REAL("gtyp_Interface_Dashboard".Publish.PosPanTiltUnit.i_degree)));
                   #ldi_StepVertical := REAL_TO_DINT("FC_Scale_linear"(inr_Y1 := DINT_TO_REAL("gtyp_SSC".Vertical_Axis.Config.di_Neg_Soft_Switch),
                                                                                                         inr_Y2 := DINT_TO_REAL("gtyp_SSC".Vertical_Axis.Config.di_Pos_Soft_Switch),
                                                                                                         inr_X1 := 0.0,
                                                                                                         inr_X2 := 180.0,
                                                                                                         inr_X := DINT_TO_REAL("gtyp_Interface_Dashboard".Publish.PosPanTiltUnit.i_degree)));
                   // Procedure - relmove_left
                   IF ("gtyp_Interface_Dashboard".Publish.PosPanTiltUnit.s_cmd = 'relmove_left')
                       AND (("gtyp_SSC".Horizontal_Axis.di_Actual_Position - #ldi_StepHorizontal) > "gtyp_SSC".Horizontal_Axis.Config.di_Neg_Soft_Switch + 15)
                       AND NOT "IX_SSC_RefSwitchHorizontalAxis_I2" THEN
                       #ldi_TargetPosition_Horizontal := "gtyp_SSC".Horizontal_Axis.di_Actual_Position - #ldi_StepHorizontal;
                       "gtyp_SSC".Horizontal_Axis.di_Target_Position := #ldi_TargetPosition_Horizontal;
                       "gtyp_SSC".Horizontal_Axis.x_Start_Positioning := TRUE;
                       #li_StepCase := 70;
                       // Procedure - relmove_right
                   ELSIF ("gtyp_Interface_Dashboard".Publish.PosPanTiltUnit.s_cmd = 'relmove_right')
                       AND (("gtyp_SSC".Horizontal_Axis.di_Actual_Position + #ldi_StepHorizontal) < "gtyp_SSC".Horizontal_Axis.Config.di_Pos_Soft_Switch - 15) THEN
                       #ldi_TargetPosition_Horizontal := "gtyp_SSC".Horizontal_Axis.di_Actual_Position + #ldi_StepHorizontal;
                       "gtyp_SSC".Horizontal_Axis.di_Target_Position := #ldi_TargetPosition_Horizontal;
                       "gtyp_SSC".Horizontal_Axis.x_Start_Positioning := TRUE;
                       #li_StepCase := 70;
                       // Procedure - relmove_up
                   ELSIF ("gtyp_Interface_Dashboard".Publish.PosPanTiltUnit.s_cmd = 'relmove_up')
                       AND (("gtyp_SSC".Vertical_Axis.di_Actual_Position + #ldi_StepHorizontal) < "gtyp_SSC".Vertical_Axis.Config.di_Pos_Soft_Switch - 15) THEN
                       #ldi_TargetPosition_Vertical := "gtyp_SSC".Vertical_Axis.di_Actual_Position + #ldi_StepVertical;
                       "gtyp_SSC".Vertical_Axis.di_Target_Position := #ldi_TargetPosition_Vertical;
                       "gtyp_SSC".Vertical_Axis.x_Start_Positioning := TRUE;
                       #li_StepCase := 80;
                       // Procedure - relmove_down
                   ELSIF ("gtyp_Interface_Dashboard".Publish.PosPanTiltUnit.s_cmd = 'relmove_down')
                       AND (("gtyp_SSC".Vertical_Axis.di_Actual_Position - #ldi_StepVertical) > "gtyp_SSC".Vertical_Axis.Config.di_Neg_Soft_Switch + 15)
                       AND NOT "IX_SSC_RefSwitchVerticalAxis_I1" THEN
                       #ldi_TargetPosition_Vertical := "gtyp_SSC".Vertical_Axis.di_Actual_Position - #ldi_StepVertical;
                       "gtyp_SSC".Vertical_Axis.di_Target_Position := #ldi_TargetPosition_Vertical;
                       "gtyp_SSC".Vertical_Axis.x_Start_Positioning := TRUE;
                       #li_StepCase := 80;
                       // Procedure - first 
                   ELSIF #lx_FirstCentre THEN
                       #li_StepCase := 20;
                       // Procedure - home
                   ELSIF ("gtyp_Interface_Dashboard".Publish.PosPanTiltUnit.s_cmd = 'home') THEN
                       #li_StepCase := 60;
                       // Procedure - start_pan
                   ELSIF ("gtyp_Interface_Dashboard".Publish.PosPanTiltUnit.s_cmd = 'start_pan')
                       AND ("gtyp_SSC".Horizontal_Axis.di_Actual_Position > "gtyp_SSC".Horizontal_Axis.Config.di_Neg_Soft_Switch + 15)
                       AND NOT "IX_SSC_RefSwitchHorizontalAxis_I2" THEN
                       #ldi_TargetPosition_Horizontal := "gtyp_SSC".Horizontal_Axis.Config.di_Neg_Soft_Switch + 15;
                       "gtyp_SSC".Horizontal_Axis.di_Target_Position := #ldi_TargetPosition_Horizontal;
                       "gtyp_SSC".Horizontal_Axis.x_Start_Positioning := TRUE;
                       #li_StepCase := 70;
                       // Procedure - end_pan
                   ELSIF ("gtyp_Interface_Dashboard".Publish.PosPanTiltUnit.s_cmd = 'end_pan')
                       AND ("gtyp_SSC".Horizontal_Axis.di_Actual_Position < "gtyp_SSC".Horizontal_Axis.Config.di_Pos_Soft_Switch - 15) THEN
                       #ldi_TargetPosition_Horizontal := "gtyp_SSC".Horizontal_Axis.Config.di_Pos_Soft_Switch - 15;
                       "gtyp_SSC".Horizontal_Axis.di_Target_Position := #ldi_TargetPosition_Horizontal;
                       "gtyp_SSC".Horizontal_Axis.x_Start_Positioning := TRUE;
                       #li_StepCase := 70;
                       // Procedure - start_tilt
                   ELSIF ("gtyp_Interface_Dashboard".Publish.PosPanTiltUnit.s_cmd = 'start_tilt')
                       AND ("gtyp_SSC".Vertical_Axis.di_Actual_Position > "gtyp_SSC".Vertical_Axis.Config.di_Neg_Soft_Switch + 15)
                       AND NOT "IX_SSC_RefSwitchVerticalAxis_I1" THEN
                       #ldi_TargetPosition_Vertical := "gtyp_SSC".Vertical_Axis.Config.di_Neg_Soft_Switch + 15;
                       "gtyp_SSC".Vertical_Axis.di_Target_Position := #ldi_TargetPosition_Vertical;
                       "gtyp_SSC".Vertical_Axis.x_Start_Positioning := TRUE;
                       #li_StepCase := 80;
                       // Procedure - end_tilt
                   ELSIF ("gtyp_Interface_Dashboard".Publish.PosPanTiltUnit.s_cmd = 'end_tilt')
                       AND ("gtyp_SSC".Vertical_Axis.di_Actual_Position < "gtyp_SSC".Vertical_Axis.Config.di_Pos_Soft_Switch - 15) THEN
                       #ldi_TargetPosition_Vertical := "gtyp_SSC".Vertical_Axis.Config.di_Pos_Soft_Switch - 15;
                       "gtyp_SSC".Vertical_Axis.di_Target_Position := #ldi_TargetPosition_Vertical;
                       "gtyp_SSC".Vertical_Axis.x_Start_Positioning := TRUE;
                       #li_StepCase := 80;
                   END_IF;
               END_IF;

           20: // homing vertical/horizontal axis
               "gtyp_SSC".Horizontal_Axis.x_Reference := TRUE;
               "gtyp_SSC".Vertical_Axis.x_Reference := TRUE;

               IF NOT "gtyp_SSC".Horizontal_Axis.x_Referenced AND NOT "gtyp_SSC".Vertical_Axis.x_Referenced THEN
                   #li_StepCase := 30;
               END_IF;

           30: // homed vertical/horizontal axis
               IF "gtyp_SSC".Horizontal_Axis.x_Referenced THEN
                   "gtyp_SSC".Horizontal_Axis.x_Reference := FALSE;
               END_IF;
               IF "gtyp_SSC".Vertical_Axis.x_Referenced THEN
                   "gtyp_SSC".Vertical_Axis.x_Reference := FALSE;
               END_IF;

               IF "gtyp_SSC".Horizontal_Axis.x_Referenced AND "gtyp_SSC".Vertical_Axis.x_Referenced THEN
                   "gtyp_SSC".Horizontal_Axis.x_Reference := FALSE;
                   "gtyp_SSC".Vertical_Axis.x_Reference := FALSE;
                   #lx_Start_TON_Wait := TRUE;
                   #li_StepCase := 40;
               END_IF;

           40: // wait sequence
               IF #lfb_TON_Wait.Q THEN
                   #lx_Start_TON_Wait := FALSE;
                   #li_StepCase := 50;
               END_IF;

           50: // Position horizontal/vertical axis and reached
               "gtyp_SSC".Horizontal_Axis.di_Target_Position := "gtyp_SSC".di_Pos_HBW_Horizontal;
               "gtyp_SSC".Horizontal_Axis.x_Start_Positioning := TRUE;
               "gtyp_SSC".Vertical_Axis.di_Target_Position := "gtyp_SSC".di_Pos_HBW_Vertical;
               "gtyp_SSC".Vertical_Axis.x_Start_Positioning := TRUE;

               IF ("gtyp_SSC".Horizontal_Axis.di_Actual_Position <= ("gtyp_SSC".di_Pos_HBW_Horizontal + "gtyp_SSC".Horizontal_Axis.Config.di_Pos_Window))
                   AND ("gtyp_SSC".Horizontal_Axis.di_Actual_Position >= ("gtyp_SSC".di_Pos_HBW_Horizontal - "gtyp_SSC".Horizontal_Axis.Config.di_Pos_Window))
                   AND "gtyp_SSC".Horizontal_Axis.x_Position_Reached THEN
                   "gtyp_SSC".Horizontal_Axis.x_Start_Positioning := FALSE;
               END_IF;

               IF ("gtyp_SSC".Vertical_Axis.di_Actual_Position <= ("gtyp_SSC".di_Pos_HBW_Vertical + "gtyp_SSC".Vertical_Axis.Config.di_Pos_Window))
                   AND ("gtyp_SSC".Vertical_Axis.di_Actual_Position >= ("gtyp_SSC".di_Pos_HBW_Vertical - "gtyp_SSC".Vertical_Axis.Config.di_Pos_Window))
                   AND "gtyp_SSC".Vertical_Axis.x_Position_Reached THEN
                   "gtyp_SSC".Vertical_Axis.x_Start_Positioning := FALSE;
               END_IF;

               IF ("gtyp_SSC".Horizontal_Axis.di_Actual_Position <= ("gtyp_SSC".di_Pos_HBW_Horizontal + "gtyp_SSC".Horizontal_Axis.Config.di_Pos_Window))
                   AND ("gtyp_SSC".Horizontal_Axis.di_Actual_Position >= ("gtyp_SSC".di_Pos_HBW_Horizontal - "gtyp_SSC".Horizontal_Axis.Config.di_Pos_Window))
                   AND "gtyp_SSC".Horizontal_Axis.x_Position_Reached
                   AND ("gtyp_SSC".Vertical_Axis.di_Actual_Position <= ("gtyp_SSC".di_Pos_HBW_Vertical + "gtyp_SSC".Vertical_Axis.Config.di_Pos_Window))
                   AND ("gtyp_SSC".Vertical_Axis.di_Actual_Position >= ("gtyp_SSC".di_Pos_HBW_Vertical - "gtyp_SSC".Vertical_Axis.Config.di_Pos_Window))
                   AND "gtyp_SSC".Vertical_Axis.x_Position_Reached THEN
                   "gtyp_SSC".Horizontal_Axis.x_Start_Positioning := FALSE;
                   "gtyp_SSC".Vertical_Axis.x_Start_Positioning := FALSE;
                   #lx_FirstCentre := FALSE;
                   #li_StepCase := 90;
               END_IF;

           60: // Position Centre horizontal/vertical axis and reached
               "gtyp_SSC".Horizontal_Axis.di_Target_Position := "gtyp_SSC".di_Pos_Centre_Horizontal;
               "gtyp_SSC".Horizontal_Axis.x_Start_Positioning := TRUE;
               "gtyp_SSC".Vertical_Axis.di_Target_Position := "gtyp_SSC".di_Pos_Centre_Vertical;
               "gtyp_SSC".Vertical_Axis.x_Start_Positioning := TRUE;

               IF ("gtyp_SSC".Horizontal_Axis.di_Actual_Position <= ("gtyp_SSC".di_Pos_Centre_Horizontal + "gtyp_SSC".Horizontal_Axis.Config.di_Pos_Window))
                   AND ("gtyp_SSC".Horizontal_Axis.di_Actual_Position >= ("gtyp_SSC".di_Pos_Centre_Horizontal - "gtyp_SSC".Horizontal_Axis.Config.di_Pos_Window))
                   AND "gtyp_SSC".Horizontal_Axis.x_Position_Reached THEN
                   "gtyp_SSC".Horizontal_Axis.x_Start_Positioning := FALSE;
               END_IF;

               IF ("gtyp_SSC".Vertical_Axis.di_Actual_Position <= ("gtyp_SSC".di_Pos_Centre_Vertical + "gtyp_SSC".Vertical_Axis.Config.di_Pos_Window))
                   AND ("gtyp_SSC".Vertical_Axis.di_Actual_Position >= ("gtyp_SSC".di_Pos_Centre_Vertical - "gtyp_SSC".Vertical_Axis.Config.di_Pos_Window))
                   AND "gtyp_SSC".Vertical_Axis.x_Position_Reached THEN
                   "gtyp_SSC".Vertical_Axis.x_Start_Positioning := FALSE;
               END_IF;

               IF ("gtyp_SSC".Horizontal_Axis.di_Actual_Position <= ("gtyp_SSC".di_Pos_Centre_Horizontal + "gtyp_SSC".Horizontal_Axis.Config.di_Pos_Window))
                   AND ("gtyp_SSC".Horizontal_Axis.di_Actual_Position >= ("gtyp_SSC".di_Pos_Centre_Horizontal - "gtyp_SSC".Horizontal_Axis.Config.di_Pos_Window))
                   AND "gtyp_SSC".Horizontal_Axis.x_Position_Reached
                   AND ("gtyp_SSC".Vertical_Axis.di_Actual_Position <= ("gtyp_SSC".di_Pos_Centre_Vertical + "gtyp_SSC".Vertical_Axis.Config.di_Pos_Window))
                   AND ("gtyp_SSC".Vertical_Axis.di_Actual_Position >= ("gtyp_SSC".di_Pos_Centre_Vertical - "gtyp_SSC".Vertical_Axis.Config.di_Pos_Window))
                   AND "gtyp_SSC".Vertical_Axis.x_Position_Reached THEN
                   "gtyp_SSC".Horizontal_Axis.x_Start_Positioning := FALSE;
                   "gtyp_SSC".Vertical_Axis.x_Start_Positioning := FALSE;
                   #lx_FirstCentre := FALSE;
                   #li_StepCase := 90;
               END_IF;

           70: // Position horizontal axis reached
               IF ("gtyp_SSC".Horizontal_Axis.di_Actual_Position <= (#ldi_TargetPosition_Horizontal + "gtyp_SSC".Horizontal_Axis.Config.di_Pos_Window))
                   AND ("gtyp_SSC".Horizontal_Axis.di_Actual_Position >= (#ldi_TargetPosition_Horizontal - "gtyp_SSC".Horizontal_Axis.Config.di_Pos_Window))
                   AND "gtyp_SSC".Horizontal_Axis.x_Position_Reached THEN
                   "gtyp_SSC".Horizontal_Axis.x_Start_Positioning := FALSE;
                   #li_StepCase := 90;
               END_IF;

           80: // Position vertical axis reached
               IF ("gtyp_SSC".Vertical_Axis.di_Actual_Position <= (#ldi_TargetPosition_Vertical + "gtyp_SSC".Vertical_Axis.Config.di_Pos_Window))
                   AND ("gtyp_SSC".Vertical_Axis.di_Actual_Position >= (#ldi_TargetPosition_Vertical - "gtyp_SSC".Vertical_Axis.Config.di_Pos_Window))
                   AND "gtyp_SSC".Vertical_Axis.x_Position_Reached THEN
                   "gtyp_SSC".Vertical_Axis.x_Start_Positioning := FALSE;
                   #li_StepCase := 90;
               END_IF;

           90: // convert the position to degrees
               "gtyp_Interface_Dashboard".Subscribe.PosPanTiltUnit.r_pan := "FC_Scale_linear"(inr_Y1 := -1.0,
                                                                                              inr_Y2 := 1.0,
                                                                                              inr_X1 := DINT_TO_REAL("gtyp_SSC".Horizontal_Axis.Config.di_Neg_Soft_Switch),
                                                                                              inr_X2 := DINT_TO_REAL("gtyp_SSC".Horizontal_Axis.Config.di_Pos_Soft_Switch),
                                                                                              inr_X := "gtyp_SSC".Horizontal_Axis.di_Actual_Position);
               "gtyp_Interface_Dashboard".Subscribe.PosPanTiltUnit.r_tilt := "FC_Scale_linear"(inr_Y1 := -1.0,
                                                                                               inr_Y2 := 1.0,
                                                                                               inr_X1 := DINT_TO_REAL("gtyp_SSC".Vertical_Axis.Config.di_Neg_Soft_Switch),
                                                                                               inr_X2 := DINT_TO_REAL("gtyp_SSC".Vertical_Axis.Config.di_Pos_Soft_Switch),
                                                                                               inr_X := "gtyp_SSC".Vertical_Axis.di_Actual_Position);

               #li_Return_write := RD_SYS_T(#ldt_write);
               "gtyp_Interface_Dashboard".Subscribe.PosPanTiltUnit.ldt_ts := DT_TO_LDT(#ldt_write);
               #lx_Start_TON_Wait := TRUE;
               #li_StepCase := 100;

           100:// wait sequence
               IF #lfb_TON_Wait.Q THEN
                   #lx_Start_TON_Wait := FALSE;
                   #li_StepCase := 0;
               END_IF;
               // Statement section ELSE        
           ELSE
               ;
       END_CASE;

   ELSE
       #lx_Init := TRUE;
       #lx_FirstCentre := TRUE;

       "gtyp_SSC".x_Start_Park_Position := FALSE;
       "gtyp_SSC".x_Park_Position_Reached := FALSE;
       "gtyp_SSC".x_Error := FALSE;
   END_IF;
END_FUNCTION_BLOCK

FUNCTION_BLOCK "PRG_SSC_Set_Positioning"   // FB13, SCL
TITLE = Program Set Positioning SSC
{ S7_Optimized_Access := 'TRUE' }
AUTHOR : A.Schaefer
VERSION : 0.0
   VAR
      lx_Init : Bool;
      lx_Start_TON_Wait : Bool;
      lx_Start_Positioning_m : Bool;
      lt_TON_Wait : Time;
      li_StepCase : Int;
      ldi_Pos_Horizontal : DInt;
      ldi_Pos_Vertical : DInt;
      lfb_R_Trig_Deaktivate : R_TRIG;
      lfb_TON_Wait : TON_TIME;
   END_VAR
BEGIN
   IF #lx_Init THEN

       // FB TON Wait
       #lfb_TON_Wait(IN := #lx_Start_TON_Wait,
                     PT := #lt_TON_Wait);

       #lfb_R_Trig_Deaktivate(CLK := NOT "gtyp_Setup".x_Set_Pos_Activ
                              OR NOT (("gtyp_Setup".i_Pos_Selection > 0)
                              AND ("gtyp_Setup".i_Pos_Selection < 21)));
       // Deaktivate step 10   
       IF #lfb_R_Trig_Deaktivate.Q THEN
           "gtyp_SSC".Horizontal_Axis.x_Start_Positioning := FALSE;
           "gtyp_SSC".Vertical_Axis.x_Start_Positioning := FALSE;
           "gtyp_SSC".Horizontal_Axis.x_Reference := FALSE;
           "gtyp_SSC".Vertical_Axis.x_Reference := FALSE;
           "gtyp_Setup".x_Start_Positioning := FALSE;
           "gtyp_Setup".x_Final_Positioning := FALSE;
           "gtyp_Setup".x_Home_Positioning := FALSE;
           "gtyp_Setup".x_Start_Offset := FALSE;
           #lx_Start_Positioning_m := FALSE;
           IF (#li_StepCase > 10) THEN
               #li_StepCase := 70;
           END_IF;
       END_IF;

       // Set Positioning activ?
       IF "gtyp_Setup".x_Set_Pos_Activ
           AND (("gtyp_Setup".i_Pos_Selection > 0)
           AND ("gtyp_Setup".i_Pos_Selection < 21))
           AND ((#li_StepCase = 40)
           OR (#li_StepCase = 60)) THEN

           // Deciding which Position
           // Position - Centre
           IF "gtyp_Setup".i_Pos_Selection = 1 THEN
               #ldi_Pos_Horizontal := "gtyp_SSC".di_Pos_Centre_Horizontal;
               #ldi_Pos_Vertical := "gtyp_SSC".di_Pos_Centre_Vertical;
               // Position - HBW 
           ELSIF "gtyp_Setup".i_Pos_Selection = 2 THEN
               #ldi_Pos_Horizontal := "gtyp_SSC".di_Pos_HBW_Horizontal;
               #ldi_Pos_Vertical := "gtyp_SSC".di_Pos_HBW_Vertical;
           END_IF;
       END_IF;

       // Set Positioning activ?
       IF NOT "gtyp_Setup".x_Set_Pos_Activ THEN
           "gtyp_Setup".i_Pos_Selection := 0;
       END_IF;

       // step chain HBW
       CASE #li_StepCase OF

           0:  // init
               #lx_Start_TON_Wait := FALSE;
               #li_StepCase := 10;

           10:  // Set Positioning activ?
               IF "gtyp_Setup".x_Set_Pos_Activ
                   AND (("gtyp_Setup".i_Pos_Selection > 0)
                   AND ("gtyp_Setup".i_Pos_Selection < 21)) THEN
                   "gtyp_SSC".Horizontal_Axis.x_Start_Positioning := FALSE;
                   "gtyp_SSC".Vertical_Axis.x_Start_Positioning := FALSE;
                   "gtyp_SSC".Horizontal_Axis.x_Reference := FALSE;
                   "gtyp_SSC".Vertical_Axis.x_Reference := FALSE;
                   "gtyp_Setup".x_Start_Positioning := FALSE;
                   "gtyp_Setup".x_Final_Positioning := FALSE;
                   "gtyp_Setup".x_Home_Positioning := FALSE;
                   "gtyp_Setup".x_Start_Offset := FALSE;
                   #li_StepCase := 20;
               END_IF;

           20: //homing vertical/horizontal axis

               "gtyp_SSC".Horizontal_Axis.x_Reference := TRUE;
               "gtyp_SSC".Vertical_Axis.x_Reference := TRUE;

               IF NOT "gtyp_SSC".Horizontal_Axis.x_Referenced AND NOT "gtyp_SSC".Vertical_Axis.x_Referenced THEN
                   #li_StepCase := 30;
               END_IF;

           30: // homed vertical/horizontal axis
               IF "gtyp_SSC".Horizontal_Axis.x_Referenced THEN
                   "gtyp_SSC".Horizontal_Axis.x_Reference := FALSE;
               END_IF;
               IF "gtyp_SSC".Vertical_Axis.x_Referenced THEN
                   "gtyp_SSC".Vertical_Axis.x_Reference := FALSE;
               END_IF;

               IF "gtyp_SSC".Horizontal_Axis.x_Referenced AND "gtyp_SSC".Vertical_Axis.x_Referenced THEN
                   "gtyp_SSC".Horizontal_Axis.x_Reference := FALSE;
                   "gtyp_SSC".Vertical_Axis.x_Reference := FALSE;
                   #li_StepCase := 40;
               END_IF;

           40:  // Start Positioning Step next
               IF "gtyp_Setup".x_Start_Positioning OR #lx_Start_Positioning_m THEN
                   #lx_Start_Positioning_m := FALSE;
                   #li_StepCase := 50;
               END_IF;

           50: // Position vertical/horizontal HBW
               "gtyp_SSC".Horizontal_Axis.di_Target_Position := #ldi_Pos_Horizontal;
               "gtyp_SSC".Horizontal_Axis.x_Start_Positioning := TRUE;
               "gtyp_SSC".Vertical_Axis.di_Target_Position := #ldi_Pos_Vertical;
               "gtyp_SSC".Vertical_Axis.x_Start_Positioning := TRUE;

               IF ("gtyp_SSC".Horizontal_Axis.di_Actual_Position <= (#ldi_Pos_Horizontal + "gtyp_SSC".Horizontal_Axis.Config.di_Pos_Window))
                   AND ("gtyp_SSC".Horizontal_Axis.di_Actual_Position >= (#ldi_Pos_Horizontal - "gtyp_SSC".Horizontal_Axis.Config.di_Pos_Window))
                   AND "gtyp_SSC".Horizontal_Axis.x_Position_Reached THEN
                   "gtyp_SSC".Horizontal_Axis.x_Start_Positioning := FALSE;
               END_IF;

               IF ("gtyp_SSC".Vertical_Axis.di_Actual_Position <= (#ldi_Pos_Vertical + "gtyp_SSC".Vertical_Axis.Config.di_Pos_Window))
                   AND ("gtyp_SSC".Vertical_Axis.di_Actual_Position >= (#ldi_Pos_Vertical - "gtyp_SSC".Vertical_Axis.Config.di_Pos_Window))
                   AND "gtyp_SSC".Vertical_Axis.x_Position_Reached THEN
                   "gtyp_SSC".Vertical_Axis.x_Start_Positioning := FALSE;
               END_IF;

               IF ("gtyp_SSC".Horizontal_Axis.di_Actual_Position <= (#ldi_Pos_Horizontal + "gtyp_SSC".Horizontal_Axis.Config.di_Pos_Window))
                   AND ("gtyp_SSC".Horizontal_Axis.di_Actual_Position >= (#ldi_Pos_Horizontal - "gtyp_SSC".Horizontal_Axis.Config.di_Pos_Window))
                   AND "gtyp_SSC".Horizontal_Axis.x_Position_Reached
                   AND ("gtyp_SSC".Vertical_Axis.di_Actual_Position <= (#ldi_Pos_Vertical + "gtyp_SSC".Vertical_Axis.Config.di_Pos_Window))
                   AND ("gtyp_SSC".Vertical_Axis.di_Actual_Position >= (#ldi_Pos_Vertical - "gtyp_SSC".Vertical_Axis.Config.di_Pos_Window))
                   AND "gtyp_SSC".Vertical_Axis.x_Position_Reached THEN
                   "gtyp_SSC".Horizontal_Axis.x_Start_Positioning := FALSE;
                   "gtyp_SSC".Vertical_Axis.x_Start_Positioning := FALSE;
                   "gtyp_Setup".x_Start_Positioning := FALSE;
                   #li_StepCase := 60;
               END_IF;

           60: // Deciding which doing

               // Start new Positioning
               IF "gtyp_Setup".x_Start_Positioning OR "gtyp_Setup".x_Home_Positioning THEN
                   #lx_Start_Positioning_m := TRUE;
                   #li_StepCase := 10;
               ELSIF #lfb_R_Trig_Deaktivate.Q THEN
                   "gtyp_Setup".x_Home_Positioning := FALSE;
                   #li_StepCase := 70;
               END_IF;

           70: //homing vertical/horizontal axis

               "gtyp_SSC".Horizontal_Axis.x_Reference := TRUE;
               "gtyp_SSC".Vertical_Axis.x_Reference := TRUE;

               IF NOT "gtyp_SSC".Horizontal_Axis.x_Referenced AND NOT "gtyp_SSC".Vertical_Axis.x_Referenced THEN
                   #li_StepCase := 80;
               END_IF;

           80: // homed vertical/horizontal axis
               IF "gtyp_SSC".Horizontal_Axis.x_Referenced THEN
                   "gtyp_SSC".Horizontal_Axis.x_Reference := FALSE;
               END_IF;
               IF "gtyp_SSC".Vertical_Axis.x_Referenced THEN
                   "gtyp_SSC".Vertical_Axis.x_Reference := FALSE;
               END_IF;

               IF "gtyp_SSC".Horizontal_Axis.x_Referenced AND "gtyp_SSC".Vertical_Axis.x_Referenced THEN
                   "gtyp_SSC".Horizontal_Axis.x_Reference := FALSE;
                   "gtyp_SSC".Vertical_Axis.x_Reference := FALSE;
                   #li_StepCase := 0;
               END_IF;

               // Statement section ELSE    
           ELSE
               ;
       END_CASE;

       IF (("gtyp_Setup".i_Pos_Selection > 0)
           AND ("gtyp_Setup".i_Pos_Selection < 21)) THEN
           // Reload Pos Value
           "gtyp_Setup".di_Pos_Horizontal := #ldi_Pos_Horizontal;
           "gtyp_Setup".di_Pos_Vertical := #ldi_Pos_Vertical;
           "gtyp_Setup".di_Pos_Rotate := 0;
       END_IF;
   ELSE
       #lx_Init := TRUE;
   END_IF;
END_FUNCTION_BLOCK

FUNCTION_BLOCK "PRG_SSC_Light"   // FB21, SCL
TITLE = Program Lights
{ S7_Optimized_Access := 'TRUE' }
AUTHOR : A.Schaefer
VERSION : 0.0
   VAR
      lx_Init : Bool;
      lx_Start : Bool;
      li_StepCase : Int;
      ldt_MQTT : Date_And_Time;
      lldt_ts_old : LDT;
      li_Return_LDT : Int;
      lfb_TOF_Camera : TOF_TIME;
      lfb_TON_Schritt : TON_TIME;
      lfb_blinker_cam : "FB_Blinker";
      lfb_blinker_config : "FB_Blinker";
      lx_StartTimer : Bool;
   END_VAR
BEGIN
   IF #lx_Init THEN

       // if camera sen picture - Red light flash
       IF "gtyp_Interface_Dashboard".Subscribe.CameraPicture.ldt_ts > #lldt_ts_old THEN
           #lldt_ts_old := "gtyp_Interface_Dashboard".Subscribe.CameraPicture.ldt_ts;
           #lfb_blinker_cam(int_periodendauer := T#50ms);
       END_IF;

       // reload flash
       "QX_SSC_LED_Red_Online_Q8" := #lfb_blinker_cam.outx_blinker;

       // FB flash config
       #lfb_blinker_config(int_periodendauer := T#500ms);

       //  Deciding which state
       //  Setup - Calibration State
       IF "gtyp_Setup".x_Set_Pos_Activ OR "gtyp_Setup".x_Color_Sensor_Calibration
           OR "gtyp_Setup".x_Counter_Value_Calibration
           OR "gtyp_Setup".x_Clean_Rack_HBW THEN
           "QX_SSC_LED_Green_Q5" := #lfb_blinker_config.outx_blinker;
           "QX_SSC_LED_Yellow_Q6" := #lfb_blinker_config.outx_blinker;
           "QX_SSC_LED_Red_Q7" := #lfb_blinker_config.outx_blinker;
           //  Error State
       ELSIF ("gtyp_Interface_Dashboard".Subscribe.State_HBW.i_code = 4)
           OR ("gtyp_Interface_Dashboard".Subscribe.State_MPO.i_code = 4)
           OR ("gtyp_Interface_Dashboard".Subscribe.State_SLD.i_code = 4)
           OR ("gtyp_Interface_Dashboard".Subscribe.State_VGR.i_code = 4) THEN
           "QX_SSC_LED_Green_Q5" := FALSE;
           "QX_SSC_LED_Yellow_Q6" := FALSE;
           "QX_SSC_LED_Red_Q7" := TRUE;
           //  Proccessing State
       ELSIF ("gtyp_Interface_Dashboard".Subscribe.State_HBW.i_code = 2)
           OR ("gtyp_Interface_Dashboard".Subscribe.State_MPO.i_code = 2)
           OR ("gtyp_Interface_Dashboard".Subscribe.State_SLD.i_code = 2)
           OR ("gtyp_Interface_Dashboard".Subscribe.State_VGR.i_code = 2) THEN
           "QX_SSC_LED_Green_Q5" := FALSE;
           "QX_SSC_LED_Yellow_Q6" := TRUE;
           "QX_SSC_LED_Red_Q7" := FALSE;
           //  Idle State
       ELSIF ("gtyp_Interface_Dashboard".Subscribe.State_HBW.i_code = 1)
           AND ("gtyp_Interface_Dashboard".Subscribe.State_MPO.i_code = 1)
           AND ("gtyp_Interface_Dashboard".Subscribe.State_SLD.i_code = 1)
           AND ("gtyp_Interface_Dashboard".Subscribe.State_VGR.i_code = 1) THEN
           "QX_SSC_LED_Green_Q5" := TRUE;
           "QX_SSC_LED_Yellow_Q6" := FALSE;
           "QX_SSC_LED_Red_Q7" := FALSE;
           //  nothing State
       ELSE
           "QX_SSC_LED_Green_Q5" := FALSE;
           "QX_SSC_LED_Yellow_Q6" := FALSE;
           "QX_SSC_LED_Red_Q7" := FALSE;
       END_IF;


   ELSE
       #lx_Init := TRUE;
   END_IF;
END_FUNCTION_BLOCK

FUNCTION_BLOCK "PRG_SSC_Axis_Horizontal"   // FB23, SCL
TITLE = Program Axis horizontal SSC
{ S7_Optimized_Access := 'TRUE' }
AUTHOR : A.Schaefer
VERSION : 0.0
   VAR
      lx_Init : Bool;
      lfb_Horizontal_Axis : "FB_Axis";
   END_VAR
BEGIN
   IF #lx_Init THEN

       // FB Axis horizontal
       #lfb_Horizontal_Axis(ini_Axis := 4,
                            indi_Increment := "gtyp_SSC".Horizontal_Axis.di_Increment,
                            inx_Ref_Switch := "IX_SSC_RefSwitchHorizontalAxis_I2",
                            inx_Referencing := "gtyp_SSC".Horizontal_Axis.x_Reference,
                            inx_Start_Positioning := "gtyp_SSC".Horizontal_Axis.x_Start_Positioning,
                            indi_Target_Position := "gtyp_SSC".Horizontal_Axis.di_Target_Position,
                            ini_PWM := "gtyp_SSC".Horizontal_Axis.i_PWM,
                            inouttyp_Config := "gtyp_SSC".Horizontal_Axis.Config,
                            inouttyp_Setup := "gtyp_SetupAxis");

       "QX_SSC_M2_HorizontalAxisCounterclockwise_Q4" := #lfb_Horizontal_Axis.outx_Motor_Neg;
       "QX_SSC_M2_HorizontalAxisClockwise_Q3" := #lfb_Horizontal_Axis.outx_Motor_Pos;
       "QW_SSC_PWM_Horizontal_M2" := #lfb_Horizontal_Axis.outi_Motor_PWM;
       "gtyp_SSC".Horizontal_Axis.di_Actual_Position := #lfb_Horizontal_Axis.outdi_Actual_Position;
       "gtyp_SSC".Horizontal_Axis.x_Referenced := #lfb_Horizontal_Axis.outx_Referenced;
       "gtyp_SSC".Horizontal_Axis.x_Position_Reached := #lfb_Horizontal_Axis.outx_Position_Reached;
   ELSE
       #lx_Init := TRUE;
   END_IF;
END_FUNCTION_BLOCK

FUNCTION_BLOCK "PRG_SSC_Axis_Horizontal_Act_Pos"   // FB24, SCL
TITLE = Program Axis horizontal Actual Position SSC
{ S7_Optimized_Access := 'TRUE' }
AUTHOR : A.Schaefer
VERSION : 0.0
   VAR
      lfb_IN_DEC : "FB_INC_DEC";
   END_VAR
BEGIN
   // FB increment axis
   #lfb_IN_DEC(inx_CHa := "IX_SSC_EncoderHorizontalAxisImp1_B3",
               inx_CHb := "IX_SSC_EncoderHorizontalAxisImp2_B4",
               ini_Ref_Wert := DINT_TO_INT("gtyp_SSC".Horizontal_Axis.Config.di_Ref_Pos),
               inx_RST := "IX_SSC_RefSwitchHorizontalAxis_I2");

   "gtyp_SSC".Horizontal_Axis.di_Increment := #lfb_IN_DEC.outi_cnt;
END_FUNCTION_BLOCK

FUNCTION_BLOCK "PRG_SSC_Axis_Vertical_Act_Pos"   // FB25, SCL
TITLE = Program Axis vertical Actual Position SSC
{ S7_Optimized_Access := 'TRUE' }
AUTHOR : A.Schaefer
VERSION : 0.0
   VAR
      lfb_IN_DEC : "FB_INC_DEC";
   END_VAR
BEGIN
   // FB increment axis
   #lfb_IN_DEC(inx_CHa := "IX_SSC_EncoderVerticalAxisImp2_B2",
               inx_CHb := "IX_SSC_EncoderVerticalAxisImp1_B1",
               ini_Ref_Wert := DINT_TO_INT("gtyp_SSC".Vertical_Axis.Config.di_Ref_Pos),
               inx_RST := "IX_SSC_RefSwitchVerticalAxis_I1");

   "gtyp_SSC".Vertical_Axis.di_Increment := #lfb_IN_DEC.outi_cnt;
END_FUNCTION_BLOCK

FUNCTION_BLOCK "PRG_SSC_Calibration_Color"   // FB32, SCL
TITLE = Program Calibration Color Sensor SSC
{ S7_Optimized_Access := 'TRUE' }
AUTHOR : A.Schaefer
VERSION : 0.0
   VAR
      lx_Init : Bool;
      lx_Start_TON_Wait : Bool;
      lx_Start_Positioning_m : Bool;
      lt_TON_Wait : Time;
      li_StepCase : Int;
      ldi_Pos_Horizontal : DInt;
      ldi_Pos_Vertical : DInt;
      lfb_R_Trig_Deaktivate : R_TRIG;
      lfb_TON_Wait : TON_TIME;
   END_VAR
BEGIN
   IF #lx_Init THEN

       // FB TON Wait
       #lfb_TON_Wait(IN := #lx_Start_TON_Wait,
                     PT := #lt_TON_Wait);

       #lfb_R_Trig_Deaktivate(CLK := NOT "gtyp_Setup".x_Color_Sensor_Calibration
                              OR NOT ("gtyp_Setup".i_Color_Sensor_Selection = 1));
       // Deaktivate step 0   
       IF #lfb_R_Trig_Deaktivate.Q THEN
           "gtyp_Setup".x_Calculate_Value_Color := FALSE;
           "gtyp_Setup".x_Set_Calib_Value_Color_Blue := FALSE;
           "gtyp_Setup".x_Set_Calib_Value_Color_Red := FALSE;
           "gtyp_Setup".x_Set_Calib_Value_Color_White := FALSE;
           "gtyp_Setup".w_Calib_ColorValue_Blue := 0;
           "gtyp_Setup".w_Calib_ColorValue_Red := 0;
           "gtyp_Setup".w_Calib_ColorValue_White := 0;
           "gtyp_Setup".w_Threshold_Red_Blue := 0;
           "gtyp_Setup".w_Threshold_White_Red := 0;
           #li_StepCase := 0;
       END_IF;

       // step chain HBW
       CASE #li_StepCase OF

           0:  // init
               #lx_Start_TON_Wait := FALSE;
               #li_StepCase := 10;

           10:  // Set Calibration activ?
               IF "gtyp_Setup".x_Color_Sensor_Calibration
                   AND ("gtyp_Setup".i_Color_Sensor_Selection = 1) THEN
                   "gtyp_Setup".x_Calculate_Value_Color := FALSE;
                   "gtyp_Setup".x_Set_Calib_Value_Color_Blue := FALSE;
                   "gtyp_Setup".x_Set_Calib_Value_Color_Red := FALSE;
                   "gtyp_Setup".x_Set_Calib_Value_Color_White := FALSE;
                   "gtyp_Setup".w_Calib_ColorValue_Blue := 0;
                   "gtyp_Setup".w_Calib_ColorValue_Red := 0;
                   "gtyp_Setup".w_Calib_ColorValue_White := 0;
                   "gtyp_Setup".w_Threshold_Red_Blue := 0;
                   "gtyp_Setup".w_Threshold_White_Red := 0;
                   #li_StepCase := 20;
               END_IF;

           20: // wait for set Values or Calculate

               // Start new Positioning
               IF "gtyp_Setup".x_Set_Calib_Value_Color_Blue THEN
                   "gtyp_Setup".w_Calib_ColorValue_Blue := "IW_SSC_ColorSensor_A1";
                   "gtyp_Setup".x_Set_Calib_Value_Color_Blue := FALSE;
               ELSIF "gtyp_Setup".x_Set_Calib_Value_Color_Red THEN
                   "gtyp_Setup".w_Calib_ColorValue_Red := "IW_SSC_ColorSensor_A1";
                   "gtyp_Setup".x_Set_Calib_Value_Color_Red := FALSE;
               ELSIF "gtyp_Setup".x_Set_Calib_Value_Color_White THEN
                   "gtyp_Setup".w_Calib_ColorValue_White := "IW_SSC_ColorSensor_A1";
                   "gtyp_Setup".x_Set_Calib_Value_Color_White := FALSE;
               END_IF;

               "gtyp_Setup".w_Threshold_White_Red := "gtyp_Setup".w_Calib_ColorValue_White + (("gtyp_Setup".w_Calib_ColorValue_Red - "gtyp_Setup".w_Calib_ColorValue_White) / 2);
               "gtyp_Setup".w_Threshold_Red_Blue := "gtyp_Setup".w_Calib_ColorValue_Red + (("gtyp_Setup".w_Calib_ColorValue_Blue - "gtyp_Setup".w_Calib_ColorValue_Red) / 2);

               IF "gtyp_Setup".x_Calculate_Value_Color THEN
                   "gtyp_SSC".w_Threshold_White_Red := "gtyp_Setup".w_Threshold_White_Red;
                   "gtyp_SSC".w_Threshold_Red_Blue := "gtyp_Setup".w_Threshold_Red_Blue;
                   "gtyp_Setup".x_Calculate_Value_Color := FALSE;
               END_IF;

               // Statement section ELSE    
           ELSE
               ;
       END_CASE;

       IF ("gtyp_Setup".i_Color_Sensor_Selection = 1) THEN
           // Reload Pos Value
           "gtyp_Setup".w_Actual_ColorValue := "IW_SSC_ColorSensor_A1";
       END_IF;
   ELSE
       #lx_Init := TRUE;
   END_IF;
END_FUNCTION_BLOCK

FUNCTION_BLOCK "PRG_SSC_Set_Park_Position"   // FB38, SCL
TITLE = Program Set Positioning SSC
{ S7_Optimized_Access := 'TRUE' }
AUTHOR : A.Schaefer
VERSION : 0.0
   VAR
      lx_Init : Bool;
      lx_Start_TON_Wait : Bool;
      lt_TON_Wait : Time;
      li_StepCase : Int;
      lfb_TON_Wait : TON_TIME;
      lfb_R_Trig_Start_Park_Pos : R_TRIG;
   END_VAR
BEGIN
   IF #lx_Init THEN

       // FB TON Wait
       #lfb_TON_Wait(IN := #lx_Start_TON_Wait,
                     PT := #lt_TON_Wait);

       #lfb_R_Trig_Start_Park_Pos(CLK := "gtyp_Setup".x_Park_Position
                                  OR "IX_Set_Park_Position");

       // Set Start Park Position   
       IF #lfb_R_Trig_Start_Park_Pos.Q THEN
           "gtyp_SSC".x_Start_Park_Position := TRUE;
           #li_StepCase := 0;
       END_IF;

       // not Start Park Pos Step 0
       IF NOT "gtyp_SSC".x_Start_Park_Position THEN
           #li_StepCase := 0;
       END_IF;

       // step chain HBW
       CASE #li_StepCase OF

           0:  // init
               #lx_Start_TON_Wait := FALSE;
               #li_StepCase := 10;

           10:  // Set Positioning activ?
               IF "gtyp_SSC".x_Start_Park_Position AND NOT "gtyp_SSC".x_Park_Position_Reached THEN
                   "gtyp_SSC".Horizontal_Axis.x_Start_Positioning := FALSE;
                   "gtyp_SSC".Vertical_Axis.x_Start_Positioning := FALSE;
                   "gtyp_SSC".Horizontal_Axis.x_Reference := FALSE;
                   "gtyp_SSC".Vertical_Axis.x_Reference := FALSE;
                   #li_StepCase := 20;
               END_IF;

           20: // homing vertical axis
               "gtyp_SSC".Vertical_Axis.x_Reference := TRUE;

               IF NOT "gtyp_SSC".Vertical_Axis.x_Referenced THEN
                   #li_StepCase := 30;
               END_IF;

           30: // homed vertical axis
               IF "gtyp_SSC".Vertical_Axis.x_Referenced THEN
                   "gtyp_SSC".Vertical_Axis.x_Reference := FALSE;
                   #li_StepCase := 40;
               END_IF;

           40: // homing horizontal axis
               "gtyp_SSC".Horizontal_Axis.x_Reference := TRUE;

               IF NOT "gtyp_SSC".Horizontal_Axis.x_Referenced THEN
                   #li_StepCase := 50;
               END_IF;

           50: // homed horizontal axis
               IF "gtyp_SSC".Horizontal_Axis.x_Referenced THEN
                   "gtyp_SSC".Horizontal_Axis.x_Reference := FALSE;
                   #li_StepCase := 60;
               END_IF;

           60: // Position horizontal Axis
               "gtyp_SSC".Horizontal_Axis.di_Target_Position := "gtyp_SSC".di_Pos_Park_Horizontal;
               "gtyp_SSC".Horizontal_Axis.x_Start_Positioning := TRUE;

               IF ("gtyp_SSC".Horizontal_Axis.di_Actual_Position <= ("gtyp_SSC".di_Pos_Park_Horizontal + "gtyp_SSC".Horizontal_Axis.Config.di_Pos_Window))
                   AND ("gtyp_SSC".Horizontal_Axis.di_Actual_Position >= ("gtyp_SSC".di_Pos_Park_Horizontal - "gtyp_SSC".Horizontal_Axis.Config.di_Pos_Window))
                   AND "gtyp_SSC".Horizontal_Axis.x_Position_Reached THEN
                   "gtyp_SSC".Horizontal_Axis.x_Start_Positioning := FALSE;
                   #li_StepCase := 70;
               END_IF;

           70: // Position vertical Axis
               "gtyp_SSC".Vertical_Axis.di_Target_Position := "gtyp_SSC".di_Pos_Park_Vertical;
               "gtyp_SSC".Vertical_Axis.x_Start_Positioning := TRUE;

               IF ("gtyp_SSC".Vertical_Axis.di_Actual_Position <= ("gtyp_SSC".di_Pos_Park_Vertical + "gtyp_SSC".Vertical_Axis.Config.di_Pos_Window))
                   AND ("gtyp_SSC".Vertical_Axis.di_Actual_Position >= ("gtyp_SSC".di_Pos_Park_Vertical - "gtyp_SSC".Vertical_Axis.Config.di_Pos_Window))
                   AND "gtyp_SSC".Vertical_Axis.x_Position_Reached THEN
                   "gtyp_SSC".Vertical_Axis.x_Start_Positioning := FALSE;
                   #li_StepCase := 80;
               END_IF;

           80: // Deciding which doing
               "gtyp_SSC".x_Park_Position_Reached := TRUE;


               // Statement section ELSE    
           ELSE
               ;
       END_CASE;

   ELSE
       #lx_Init := TRUE;
   END_IF;
END_FUNCTION_BLOCK

// folder: Tracking

FUNCTION_BLOCK "SLD_Tracking"   // FB6, SCL
{ S7_Optimized_Access := 'TRUE' }
VERSION : 0.1
   VAR
      Location : String;
   END_VAR
BEGIN

   IF NOT "IX_SLD_LightBarrierInlet_I2" THEN
       #Location := 'LightB_Inlet'; //Change value of string when lightbarier is active
       "gtyp_Interface_Dashboard".Subscribe.State_Track.track_puck := 'LightB_Inlet'; //Publish location to Node-Red
   END_IF;

   IF NOT "IX_SLD_LightBarrierBehindColorSensor_I3" THEN
       #Location := 'LightB_BehindColorSensor';
       "gtyp_Interface_Dashboard".Subscribe.State_Track.track_puck := 'LightB_BehindColorSensor';
   END_IF;

   IF NOT "IX_SLD_LightBarrierWhite_I5" THEN
       #Location := 'Light_White';
       "gtyp_Interface_Dashboard".Subscribe.State_Track.track_puck := 'LightB_White';
   END_IF;

   IF NOT "IX_SLD_LightBarrierRed_I6" THEN
       #Location := 'LightB_Red';
       "gtyp_Interface_Dashboard".Subscribe.State_Track.track_puck := 'LightB_Red';
   END_IF;

   IF NOT "IX_SLD_LightBarrierBlue_I7" THEN
       #Location := 'LightB_Blue';
       "gtyp_Interface_Dashboard".Subscribe.State_Track.track_puck := 'LightB_Blue';
   END_IF;
END_FUNCTION_BLOCK

FUNCTION_BLOCK "HBW_Tracking"   // FB42, SCL
{ S7_Optimized_Access := 'TRUE' }
VERSION : 0.1
   VAR
      Location : String;
   END_VAR
BEGIN
   //Change value of string when lightbarier is active
   IF NOT "IX_HBW_LightBarrierInside_I2" THEN
       #Location := 'LightB_Inside';
       "gtyp_Interface_Dashboard".Subscribe.State_Track.track_puck := 'LightB_Inside';
   END_IF;

   IF NOT "IX_HBW_LightBarrierOutside_I3" THEN
       #Location := 'LightB_Outside';
       "gtyp_Interface_Dashboard".Subscribe.State_Track.track_puck := 'LightB_Outside';
   END_IF;
END_FUNCTION_BLOCK

FUNCTION_BLOCK "SSC_Tracking"   // FB43, SCL
{ S7_Optimized_Access := 'TRUE' }
VERSION : 0.1
   VAR
      Location : String;
   END_VAR
BEGIN
   //Change value of string when lightbarier is active
   IF NOT "IX_SSC_LightBarrierStorage_I3" THEN
       #Location := 'LightB_Storage';
       "gtyp_Interface_Dashboard".Subscribe.State_Track.track_puck := 'LightB_Storage';
   END_IF;

   IF NOT "IX_SSC_LightBarrierOutsourcing_I4" THEN
       #Location := 'LightB_Outsourcing';
       "gtyp_Interface_Dashboard".Subscribe.State_Track.track_puck := 'LightB_Outsourcing';
   END_IF;
END_FUNCTION_BLOCK

FUNCTION_BLOCK "MPO_Tracking"   // FB44, SCL
{ S7_Optimized_Access := 'TRUE' }
VERSION : 0.1
   VAR
      Location : String;
   END_VAR
BEGIN
   //Change value of string when lightbarier is active
   IF NOT "IX_MPO_LightBarrierEndOfConBelt_I3" THEN
       #Location := 'LightB_EndBelt';
       "gtyp_Interface_Dashboard".Subscribe.State_Track.track_puck := 'LightB_EndBelt';
   END_IF;


   IF NOT "IX_MPO_LightBarrierOven_I9" THEN
       #Location := 'LightB_Oven';
       "gtyp_Interface_Dashboard".Subscribe.State_Track.track_puck := 'LightB_Oven';
   END_IF;


   //Object is outside of oven
   IF  "QX_MPO_M5_VacuumTowardsOven_Q7" OR "QX_MPO_M5_VacuumTowardsTurnTable_Q8" THEN
           #Location := 'OutsidePath';
           "gtyp_Interface_Dashboard".Subscribe.State_Track.track_puck := 'OutsidePath';
   END_IF;
END_FUNCTION_BLOCK

// folder: VGR_Vacuum_Gripper_Robot

FUNCTION_BLOCK "PRG_VGR_Axis_vertical"   // FB1, SCL
TITLE = Program Axis vertical VGR
{ S7_Optimized_Access := 'TRUE' }
AUTHOR : A.Schaefer
VERSION : 0.0
   VAR
      lx_Init : Bool;
      lfb_vertical_Axis : "FB_Axis_Auto";
   END_VAR
BEGIN
   IF #lx_Init THEN

       // FB Axis vertical
       #lfb_vertical_Axis(ini_Axis := 2,
                          indi_Increment := "gtyp_VGR".vertical_Axis.di_Increment,
                          inx_Ref_Switch := "IX_VGR_RefSwitchVerticalAxis_I1",
                          inx_Referencing := "gtyp_VGR".vertical_Axis.x_Reference,
                          inx_Start_Positioning := "gtyp_VGR".vertical_Axis.x_Start_Positioning,
                          indi_Target_Position := "gtyp_VGR".vertical_Axis.di_Target_Position,
                          ini_PWM := "gtyp_VGR".vertical_Axis.i_PWM,
                          inouttyp_Config := "gtyp_VGR".vertical_Axis.Config,
                          inouttyp_Setup := "gtyp_SetupAxis");

       "QX_VGR_M1_VerticalAxisUp_Q1" := #lfb_vertical_Axis.outx_Motor_Neg;
       "QX_VGR_M1_VerticalAxisDown_Q2" := #lfb_vertical_Axis.outx_Motor_Pos;
       "QW_VGR_PWM_Vertical_M1" := #lfb_vertical_Axis.outi_Motor_PWM;
       "gtyp_VGR".vertical_Axis.di_Actual_Position := #lfb_vertical_Axis.outdi_Actual_Position;
       "gtyp_VGR".vertical_Axis.x_Referenced := #lfb_vertical_Axis.outx_Referenced;
       "gtyp_VGR".vertical_Axis.x_Position_Reached := #lfb_vertical_Axis.outx_Position_Reached;
   ELSE
       #lx_Init := TRUE;
   END_IF;
END_FUNCTION_BLOCK

FUNCTION_BLOCK "PRG_VGR_Axis_horizontal"   // FB4, SCL
TITLE = Program Axis horizontal VGR
{ S7_Optimized_Access := 'TRUE' }
AUTHOR : A.Schaefer
VERSION : 0.0
   VAR
      lx_Init : Bool;
      lfb_horizontal_Axis : "FB_Axis_Auto";
   END_VAR
BEGIN
   IF #lx_Init THEN

       // FB Axis horizontal
       #lfb_horizontal_Axis(ini_Axis := 1,
                            indi_Increment := "gtyp_VGR".horizontal_Axis.di_Increment,
                            inx_Ref_Switch := "IX_VGR_RefSwitchHorizontalAxis_I2",
                            inx_Referencing := "gtyp_VGR".horizontal_Axis.x_Reference,
                            inx_Start_Positioning := "gtyp_VGR".horizontal_Axis.x_Start_Positioning,
                            indi_Target_Position := "gtyp_VGR".horizontal_Axis.di_Target_Position,
                            ini_PWM := "gtyp_VGR".horizontal_Axis.i_PWM,
                            inouttyp_Config := "gtyp_VGR".horizontal_Axis.Config,
                            inouttyp_Setup := "gtyp_SetupAxis");

       "QX_VGR_M2_HorizontalAxisForward_Q4" := #lfb_horizontal_Axis.outx_Motor_Pos;
       "QX_VGR_M2_HorizontalAxisBackward_Q3" := #lfb_horizontal_Axis.outx_Motor_Neg;
       "QW_VGR_PWM_Horizontal_M2" := #lfb_horizontal_Axis.outi_Motor_PWM;
       "gtyp_VGR".horizontal_Axis.di_Actual_Position := #lfb_horizontal_Axis.outdi_Actual_Position;
       "gtyp_VGR".horizontal_Axis.x_Referenced := #lfb_horizontal_Axis.outx_Referenced;
       "gtyp_VGR".horizontal_Axis.x_Position_Reached := #lfb_horizontal_Axis.outx_Position_Reached;
   ELSE
       #lx_Init := TRUE;
   END_IF;
END_FUNCTION_BLOCK

FUNCTION_BLOCK "PRG_VGR_Axis_rotate"   // FB5, SCL
TITLE = Program Axis rotate VGR
{ S7_Optimized_Access := 'TRUE' }
AUTHOR : A.Schaefer
VERSION : 0.0
   VAR
      lx_Init : Bool;
      lfb_rotate_Axis : "FB_Axis_Auto";
   END_VAR
BEGIN
   IF #lx_Init THEN

       // FB Axis rotate
       #lfb_rotate_Axis(ini_Axis := 3,
                        indi_Increment := "gtyp_VGR".rotate_Axis.di_Increment,
                        inx_Ref_Switch := "IX_VGR_RefSwitchRotate_I3",
                        inx_Referencing := "gtyp_VGR".rotate_Axis.x_Reference,
                        inx_Start_Positioning := "gtyp_VGR".rotate_Axis.x_Start_Positioning,
                        indi_Target_Position := "gtyp_VGR".rotate_Axis.di_Target_Position,
                        ini_PWM := "gtyp_VGR".rotate_Axis.i_PWM,
                        inouttyp_Config := "gtyp_VGR".rotate_Axis.Config,
                        inouttyp_Setup := "gtyp_SetupAxis");

       "QX_VGR_M3_RotateClockwise_Q5" := #lfb_rotate_Axis.outx_Motor_Neg;
       "QX_VGR_M3_RotateCounterclockwise_Q6" := #lfb_rotate_Axis.outx_Motor_Pos;
       "QW_VGR_PWM_Rotate_M3" := #lfb_rotate_Axis.outi_Motor_PWM;
       "gtyp_VGR".rotate_Axis.di_Actual_Position := #lfb_rotate_Axis.outdi_Actual_Position;
       "gtyp_VGR".rotate_Axis.x_Referenced := #lfb_rotate_Axis.outx_Referenced;
       "gtyp_VGR".rotate_Axis.x_Position_Reached := #lfb_rotate_Axis.outx_Position_Reached;
   ELSE
       #lx_Init := TRUE;
   END_IF;
END_FUNCTION_BLOCK

FUNCTION_BLOCK "PRG_VGR_Ablauf"   // FB7, SCL
TITLE = Program Ablauf VGR
{ S7_Optimized_Access := 'TRUE' }
AUTHOR : A.Schaefer
VERSION : 0.0
   VAR
      lx_Init : Bool;
      lx_Start_TON_Wait : Bool;
      lx_Start_TON_State : Bool;
      lt_TON_Wait : Time;
      ldt_MQTT : Date_And_Time;
      li_Return_LDT : Int;
      li_Lights : Int;
      li_Lights_old : Int;
      lx_State_activ : Bool;
      li_StepCase : Int;
      ldi_Pos_SLD_X : DInt;
      ldi_Pos_SLD_Y : DInt;
      ldi_Pos_SLD_Z : DInt;
      ls_Color : String;
      ls_Target : String;
      lfb_TON_Wait : TON_TIME;
      lfb_TON_State : TON_TIME;
      lfb_R_Trig_NiO : R_TRIG;
   END_VAR
   VAR_TEMP
      ti_Counter : Int;
   END_VAR
BEGIN
   IF #lx_Init THEN

       // Restart after set Positioning
       IF "gtyp_Setup".x_Set_Pos_Activ OR "gtyp_Setup".x_Color_Sensor_Calibration OR "gtyp_VGR".x_Start_Park_Position OR "gtyp_MPO".x_Error THEN
           IF "gtyp_MPO".x_Error THEN
               "gtyp_VGR".x_MPO_Req_Discard := FALSE;
               "gtyp_VGR".x_MPO_Discards := FALSE;
           END_IF;
           #li_StepCase := 0;
       END_IF;

       // wait time state
       #lfb_TON_State(IN := NOT #lx_Start_TON_State,
                      PT := T#2s);

       IF "gtyp_VGR".x_State_Process THEN
           #li_Return_LDT := RD_SYS_T(#ldt_MQTT);
           "gtyp_Interface_Dashboard".Subscribe.State_Order.ldt_ts := DT_TO_LDT(#ldt_MQTT);
       END_IF;

       // state of the robot cyclically transmitted to the cloud
       IF (#lfb_TON_State.Q OR (#li_Lights <> #li_Lights_old)) AND NOT #lx_Start_TON_State THEN
           #li_Lights_old := #li_Lights;
           #lx_Start_TON_State := TRUE;
           #li_Return_LDT := RD_SYS_T(#ldt_MQTT);
           "gtyp_Interface_Dashboard".Subscribe.State_VGR.ldt_ts := DT_TO_LDT(#ldt_MQTT);
           "gtyp_Interface_Dashboard".Subscribe.State_VGR.i_code := #li_Lights;
           "gtyp_Interface_Dashboard".Subscribe.State_VGR.s_description := '';
           "gtyp_Interface_Dashboard".Subscribe.State_VGR.s_station := 'vgr';
           "gtyp_Interface_Dashboard".Subscribe.State_VGR.s_target := #ls_Target;
           "gtyp_Interface_Dashboard".Subscribe.State_VGR.x_active := #lx_State_activ;

           "gtyp_Interface_Dashboard".Subscribe.PosPanTiltUnit.ldt_ts := DT_TO_LDT(#ldt_MQTT);

           "gtyp_Interface_Dashboard".Subscribe.State_VGR.Workpiece := "gtyp_VGR".Workpiece;
       END_IF;

       // restart wait time state
       IF NOT #lfb_TON_State.Q AND #lx_Start_TON_State THEN
           #lx_Start_TON_State := FALSE;
       END_IF;

       // rising edge Workpiece NiO
       #lfb_R_Trig_NiO(CLK := "gtyp_VGR".x_Workpiece_NiO);

       IF #lfb_R_Trig_NiO.Q THEN
           #lx_Start_TON_Wait := FALSE;
           #lx_State_activ := FALSE;
           #li_Lights := 4;
           #ls_Target := '';
           "gtyp_VGR".horizontal_Axis.x_Start_Positioning := FALSE;
           "gtyp_VGR".vertical_Axis.x_Start_Positioning := FALSE;
           "gtyp_VGR".rotate_Axis.x_Start_Positioning := FALSE;
           "gtyp_VGR".x_NFC_Start_First := FALSE;
           "gtyp_VGR".x_NFC_Start := FALSE;
           #li_StepCase := 70;
       END_IF;

       // FB TON Wait
       #lfb_TON_Wait(IN := #lx_Start_TON_Wait,
                     PT := #lt_TON_Wait);

       // step chain VGR
       CASE #li_StepCase OF

           0:  // init
               #lx_Start_TON_Wait := FALSE;
               #li_Lights := 1;
               #lx_State_activ := FALSE;
               #ls_Target := '';
               "gtyp_VGR".horizontal_Axis.x_Start_Positioning := FALSE;
               "gtyp_VGR".vertical_Axis.x_Start_Positioning := FALSE;
               "gtyp_VGR".rotate_Axis.x_Start_Positioning := FALSE;
               "gtyp_VGR".x_HBW_Storage := FALSE;
               "gtyp_VGR".x_HBW_Outsource := FALSE;
               "gtyp_VGR".x_NFC_Start_First := FALSE;
               "gtyp_VGR".x_NFC_Start := FALSE;
               "gtyp_VGR".x_Ready_For_Outsource := FALSE;
               "QX_VGR_Compressor_Q7" := FALSE;
               "QX_VGR_ValveVacuum_Q8" := FALSE;
               "gtyp_VGR".vertical_Axis.i_PWM := -1;
               "gtyp_VGR".horizontal_Axis.i_PWM := -1;
               "gtyp_VGR".rotate_Axis.i_PWM := -1;

               IF NOT "gtyp_Setup".x_Set_Pos_Activ AND NOT "gtyp_VGR".x_Start_Park_Position AND NOT "gtyp_MPO".x_Error THEN
                   #li_StepCase := 10;
               END_IF;

           10: // homing vertical axis
               #li_Lights := 2;
               "gtyp_VGR".x_Ready_For_Outsource := TRUE;
               "gtyp_VGR".vertical_Axis.x_Reference := TRUE;
               //"gtyp_VGR".vertical_Axis.i_PWM := 800;

               IF NOT "gtyp_VGR".vertical_Axis.x_Referenced THEN
                   #li_StepCase := 20;
               END_IF;

           20: // homed vertical axis
               IF "gtyp_VGR".vertical_Axis.x_Referenced THEN
                   "gtyp_VGR".vertical_Axis.x_Reference := FALSE;
                   #li_StepCase := 30;
               END_IF;

           30: // homing horizontal axis
               "gtyp_VGR".horizontal_Axis.x_Reference := TRUE;

               IF NOT "gtyp_VGR".horizontal_Axis.x_Referenced THEN
                   #li_StepCase := 40;
               END_IF;

           40: // homed horizontal axis
               IF "gtyp_VGR".horizontal_Axis.x_Referenced THEN
                   "gtyp_VGR".horizontal_Axis.x_Reference := FALSE;
                   #li_StepCase := 50;
               END_IF;

           50: // homing rotate axis
               "gtyp_VGR".rotate_Axis.x_Reference := TRUE;

               IF NOT "gtyp_VGR".rotate_Axis.x_Referenced THEN
                   #li_StepCase := 60;
               END_IF;

           60: // homed rotate axis
               IF "gtyp_VGR".rotate_Axis.x_Referenced THEN
                   "gtyp_VGR".rotate_Axis.x_Reference := FALSE;
                   #li_StepCase := 70;
               END_IF;

           70: // Deciding which route to take

               #li_Lights := 1;
               #lx_State_activ := FALSE;
               #ls_Target := '';
               "gtyp_VGR".x_Ready_For_Outsource := TRUE;

               // Procedure - bad part
               IF "gtyp_VGR".x_Workpiece_NiO THEN
                   "gtyp_VGR".x_Ready_For_Outsource := FALSE;
                   #li_Lights := 4;
                   #li_StepCase := 1200;
                   // Procedure - pick up finished parts blue
               ELSIF NOT "IX_SLD_LightBarrierBlue_I7" THEN
                   #ldi_Pos_SLD_X := "gtyp_VGR".di_Pos_SLD_Blue_horizontal;
                   #ldi_Pos_SLD_Y := "gtyp_VGR".di_Pos_SLD_Blue_vertical;
                   #ldi_Pos_SLD_Z := "gtyp_VGR".di_Pos_SLD_Blue_rotate;
                   "gtyp_VGR".x_Ready_For_Outsource := FALSE;
                   #li_StepCase := 100;
                   // Procedure - pick up finished parts red
               ELSIF NOT "IX_SLD_LightBarrierRed_I6" THEN
                   #ldi_Pos_SLD_X := "gtyp_VGR".di_Pos_SLD_Red_horizontal;
                   #ldi_Pos_SLD_Y := "gtyp_VGR".di_Pos_SLD_Red_vertical;
                   #ldi_Pos_SLD_Z := "gtyp_VGR".di_Pos_SLD_Red_rotate;
                   "gtyp_VGR".x_Ready_For_Outsource := FALSE;
                   #li_StepCase := 100;
                   // Procedure - pick up finished parts white
               ELSIF NOT "IX_SLD_LightBarrierWhite_I5" THEN
                   #ldi_Pos_SLD_X := "gtyp_VGR".di_Pos_SLD_White_horizontal;
                   #ldi_Pos_SLD_Y := "gtyp_VGR".di_Pos_SLD_White_vertical;
                   #ldi_Pos_SLD_Z := "gtyp_VGR".di_Pos_SLD_White_rotate;
                   "gtyp_VGR".x_Ready_For_Outsource := FALSE;
                   #li_StepCase := 100;
                   // Procedure - outsource to manufacturing
               ELSIF "gtyp_VGR".x_HBW_Outsource THEN
                   // Order State
                   "gtyp_Interface_Dashboard".Subscribe.State_Order.ldt_ts := DT_TO_LDT(#ldt_MQTT);
                   "gtyp_Interface_Dashboard".Subscribe.State_Order.s_state := 'ORDERED';
                   "gtyp_Interface_Dashboard".Subscribe.State_Order.s_type := "gtyp_VGR".s_HBW_Outsource_Typ;
                   #li_StepCase := 400;
                   // Procedure - store raw parts
               ELSIF (NOT "IX_SSC_LightBarrierStorage_I3") AND ("gtyp_HBW".i_Blue_Available + "gtyp_HBW".i_Red_Available + "gtyp_HBW".i_White_Available < 9) THEN
                   "gtyp_VGR".x_Ready_For_Outsource := FALSE;
                   #li_Lights := 2;
                   "gtyp_VGR".x_HBW_Storage := TRUE;
                   #li_StepCase := 600;
               END_IF;

               (**************************************************************************************************)
               (****************************    Procedure - pick up finished parts    ****************************)
               (**************************************************************************************************)
           100: // Position of finished part 

               #li_Lights := 2;
               "gtyp_VGR".horizontal_Axis.di_Target_Position := #ldi_Pos_SLD_X;
               "gtyp_VGR".horizontal_Axis.x_Start_Positioning := TRUE;

               "gtyp_VGR".vertical_Axis.x_Reference := TRUE;
               //"gtyp_VGR".vertical_Axis.i_PWM := 800;

               "gtyp_VGR".rotate_Axis.di_Target_Position := #ldi_Pos_SLD_Z;
               "gtyp_VGR".rotate_Axis.x_Start_Positioning := TRUE;

               IF ("gtyp_VGR".horizontal_Axis.di_Actual_Position <= (#ldi_Pos_SLD_X + "gtyp_VGR".horizontal_Axis.Config.di_Pos_Window))
                   AND ("gtyp_VGR".horizontal_Axis.di_Actual_Position >= (#ldi_Pos_SLD_X - "gtyp_VGR".horizontal_Axis.Config.di_Pos_Window))
                   AND "gtyp_VGR".horizontal_Axis.x_Position_Reached THEN
                   "gtyp_VGR".horizontal_Axis.x_Start_Positioning := FALSE;
               END_IF;

               IF ("gtyp_VGR".rotate_Axis.di_Actual_Position <= (#ldi_Pos_SLD_Z + "gtyp_VGR".rotate_Axis.Config.di_Pos_Window))
                   AND ("gtyp_VGR".rotate_Axis.di_Actual_Position >= (#ldi_Pos_SLD_Z - "gtyp_VGR".rotate_Axis.Config.di_Pos_Window))
                   AND "gtyp_VGR".rotate_Axis.x_Position_Reached THEN
                   "gtyp_VGR".rotate_Axis.x_Start_Positioning := FALSE;
               END_IF;

               IF NOT "gtyp_VGR".vertical_Axis.x_Referenced THEN
                   #li_StepCase := 110;
               END_IF;

           110: // position of finished part reached         

               IF ("gtyp_VGR".horizontal_Axis.di_Actual_Position <= (#ldi_Pos_SLD_X + "gtyp_VGR".horizontal_Axis.Config.di_Pos_Window))
                   AND ("gtyp_VGR".horizontal_Axis.di_Actual_Position >= (#ldi_Pos_SLD_X - "gtyp_VGR".horizontal_Axis.Config.di_Pos_Window))
                   AND "gtyp_VGR".horizontal_Axis.x_Position_Reached THEN
                   "gtyp_VGR".horizontal_Axis.x_Start_Positioning := FALSE;
               END_IF;

               IF ("gtyp_VGR".rotate_Axis.di_Actual_Position <= (#ldi_Pos_SLD_Z + "gtyp_VGR".rotate_Axis.Config.di_Pos_Window))
                   AND ("gtyp_VGR".rotate_Axis.di_Actual_Position >= (#ldi_Pos_SLD_Z - "gtyp_VGR".rotate_Axis.Config.di_Pos_Window))
                   AND "gtyp_VGR".rotate_Axis.x_Position_Reached THEN
                   "gtyp_VGR".rotate_Axis.x_Start_Positioning := FALSE;
               END_IF;

               IF "gtyp_VGR".vertical_Axis.x_Referenced THEN
                   "gtyp_VGR".vertical_Axis.x_Reference := FALSE;
               END_IF;

               IF ("gtyp_VGR".horizontal_Axis.di_Actual_Position <= (#ldi_Pos_SLD_X + "gtyp_VGR".horizontal_Axis.Config.di_Pos_Window))
                   AND ("gtyp_VGR".horizontal_Axis.di_Actual_Position >= (#ldi_Pos_SLD_X - "gtyp_VGR".horizontal_Axis.Config.di_Pos_Window))
                   AND "gtyp_VGR".horizontal_Axis.x_Position_Reached
                   AND "gtyp_VGR".vertical_Axis.x_Referenced
                   AND ("gtyp_VGR".rotate_Axis.di_Actual_Position <= (#ldi_Pos_SLD_Z + "gtyp_VGR".rotate_Axis.Config.di_Pos_Window))
                   AND ("gtyp_VGR".rotate_Axis.di_Actual_Position >= (#ldi_Pos_SLD_Z - "gtyp_VGR".rotate_Axis.Config.di_Pos_Window))
                   AND "gtyp_VGR".rotate_Axis.x_Position_Reached THEN
                   "gtyp_VGR".horizontal_Axis.x_Start_Positioning := FALSE;
                   "gtyp_VGR".vertical_Axis.x_Start_Positioning := FALSE;
                   "gtyp_VGR".rotate_Axis.x_Start_Positioning := FALSE;
                   #li_StepCase := 120;
               END_IF;

           120: // wait sequence
               #lx_Start_TON_Wait := TRUE;
               #lt_TON_Wait := T#500ms;

               IF #lfb_TON_Wait.Q THEN
                   #lx_Start_TON_Wait := FALSE;
                   #li_StepCase := 130;
               END_IF;

           130: // Position vertical finished part
               "gtyp_VGR".vertical_Axis.di_Target_Position := #ldi_Pos_SLD_Y;
               "gtyp_VGR".vertical_Axis.x_Start_Positioning := TRUE;
               //"gtyp_VGR".vertical_Axis.i_PWM := 500;

               IF ("gtyp_VGR".vertical_Axis.di_Actual_Position <= (#ldi_Pos_SLD_Y + "gtyp_VGR".vertical_Axis.Config.di_Pos_Window))
                   AND ("gtyp_VGR".vertical_Axis.di_Actual_Position >= (#ldi_Pos_SLD_Y - "gtyp_VGR".vertical_Axis.Config.di_Pos_Window))
                   AND "gtyp_VGR".vertical_Axis.x_Position_Reached THEN
                   "gtyp_VGR".vertical_Axis.x_Start_Positioning := FALSE;
                   #li_StepCase := 140;
               END_IF;

           140: // start compressor
               "QX_VGR_Compressor_Q7" := TRUE;

               #lx_Start_TON_Wait := TRUE;
               #lt_TON_Wait := T#1000ms;

               IF #lfb_TON_Wait.Q THEN
                   #lx_Start_TON_Wait := FALSE;
                   #li_StepCase := 150;
               END_IF;

           150: // turn on the vacuum and pick up the part
               "QX_VGR_ValveVacuum_Q8" := true;

               #lx_Start_TON_Wait := TRUE;
               #lt_TON_Wait := T#1000ms;

               IF #lfb_TON_Wait.Q THEN
                   #lx_Start_TON_Wait := FALSE;
                   #lx_State_activ := TRUE;
                   #ls_Target := 'dso';
                   "gtyp_VGR".History := "gtyp_SLD".History;
                   "gtyp_VGR".Workpiece := "gtyp_SLD".Workpiece;
                   "gtyp_SLD".Workpiece.s_id := '0';
                   "gtyp_SLD".Workpiece.s_state := '';
                   "gtyp_SLD".Workpiece.s_type := '';
                   FOR #ti_Counter := 1 TO 8 DO
                       "gtyp_SLD".History[#ti_Counter].i_code := 0;
                       "gtyp_SLD".History[#ti_Counter].ldt_ts := DT#1990-01-01-00:00:00;
                   END_FOR;

                   #li_Return_LDT := RD_SYS_T(#ldt_MQTT);
                   "gtyp_VGR".History[8].i_code := 800;
                   "gtyp_VGR".History[8].ldt_ts := DT_TO_LDT(#ldt_MQTT);

                   "gtyp_Interface_Dashboard".Subscribe.State_SLD.x_active := FALSE;

                   #li_StepCase := 160;
               END_IF;

           160: // Position vertical preposition NFC
               "gtyp_VGR".vertical_Axis.di_Target_Position := "gtyp_VGR".di_Pos_NFC_vertical - "gtyp_VGR".di_Offset_Pos_DSI_NFC_vertical;
               "gtyp_VGR".vertical_Axis.x_Start_Positioning := TRUE;
               //"gtyp_VGR".vertical_Axis.i_PWM := 800;

               IF ("gtyp_VGR".vertical_Axis.di_Actual_Position <= ("gtyp_VGR".di_Pos_NFC_vertical - "gtyp_VGR".di_Offset_Pos_DSI_NFC_vertical + "gtyp_VGR".vertical_Axis.Config.di_Pos_Window))
                   AND ("gtyp_VGR".vertical_Axis.di_Actual_Position >= ("gtyp_VGR".di_Pos_NFC_vertical - "gtyp_VGR".di_Offset_Pos_DSI_NFC_vertical - "gtyp_VGR".vertical_Axis.Config.di_Pos_Window))
                   AND "gtyp_VGR".vertical_Axis.x_Position_Reached THEN
                   "gtyp_VGR".vertical_Axis.x_Start_Positioning := FALSE;
                   #li_StepCase := 170;
               END_IF;

           170: // homing horizontal axis
               "gtyp_VGR".horizontal_Axis.x_Reference := TRUE;

               IF NOT "gtyp_VGR".horizontal_Axis.x_Referenced THEN
                   #li_StepCase := 180;
               END_IF;

           180: // homed horizontal axis
               IF "gtyp_VGR".horizontal_Axis.x_Referenced THEN
                   "gtyp_VGR".horizontal_Axis.x_Reference := FALSE;
                   #li_StepCase := 190;
               END_IF;

           190: // wait sequence
               #lx_Start_TON_Wait := TRUE;
               #lt_TON_Wait := T#500ms;

               IF #lfb_TON_Wait.Q THEN
                   #lx_Start_TON_Wait := FALSE;
                   #li_StepCase := 200;
               END_IF;

           200: // Position horizontal/rotate NFC

               "gtyp_VGR".horizontal_Axis.di_Target_Position := "gtyp_VGR".di_Pos_NFC_horizontal;
               "gtyp_VGR".horizontal_Axis.x_Start_Positioning := TRUE;
               "gtyp_VGR".rotate_Axis.di_Target_Position := "gtyp_VGR".di_Pos_NFC_rotate;
               "gtyp_VGR".rotate_Axis.x_Start_Positioning := TRUE;

               IF ("gtyp_VGR".horizontal_Axis.di_Actual_Position <= ("gtyp_VGR".di_Pos_NFC_horizontal + "gtyp_VGR".horizontal_Axis.Config.di_Pos_Window))
                   AND ("gtyp_VGR".horizontal_Axis.di_Actual_Position >= ("gtyp_VGR".di_Pos_NFC_horizontal - "gtyp_VGR".horizontal_Axis.Config.di_Pos_Window))
                   AND "gtyp_VGR".horizontal_Axis.x_Position_Reached THEN
                   "gtyp_VGR".horizontal_Axis.x_Start_Positioning := FALSE;
               END_IF;

               IF ("gtyp_VGR".rotate_Axis.di_Actual_Position <= ("gtyp_VGR".di_Pos_NFC_rotate + "gtyp_VGR".rotate_Axis.Config.di_Pos_Window))
                   AND ("gtyp_VGR".rotate_Axis.di_Actual_Position >= ("gtyp_VGR".di_Pos_NFC_rotate - "gtyp_VGR".rotate_Axis.Config.di_Pos_Window))
                   AND "gtyp_VGR".rotate_Axis.x_Position_Reached THEN
                   "gtyp_VGR".rotate_Axis.x_Start_Positioning := FALSE;
               END_IF;

               IF ("gtyp_VGR".horizontal_Axis.di_Actual_Position <= ("gtyp_VGR".di_Pos_NFC_horizontal + "gtyp_VGR".horizontal_Axis.Config.di_Pos_Window))
                   AND ("gtyp_VGR".horizontal_Axis.di_Actual_Position >= ("gtyp_VGR".di_Pos_NFC_horizontal - "gtyp_VGR".horizontal_Axis.Config.di_Pos_Window))
                   AND "gtyp_VGR".horizontal_Axis.x_Position_Reached
                   AND ("gtyp_VGR".rotate_Axis.di_Actual_Position <= ("gtyp_VGR".di_Pos_NFC_rotate + "gtyp_VGR".rotate_Axis.Config.di_Pos_Window))
                   AND ("gtyp_VGR".rotate_Axis.di_Actual_Position >= ("gtyp_VGR".di_Pos_NFC_rotate - "gtyp_VGR".rotate_Axis.Config.di_Pos_Window))
                   AND "gtyp_VGR".rotate_Axis.x_Position_Reached THEN
                   "gtyp_VGR".horizontal_Axis.x_Start_Positioning := FALSE;
                   "gtyp_VGR".rotate_Axis.x_Start_Positioning := FALSE;
                   #li_StepCase := 210;
               END_IF;

           210: // wait sequence
               #lx_Start_TON_Wait := TRUE;
               #lt_TON_Wait := T#500ms;

               IF #lfb_TON_Wait.Q THEN
                   #lx_Start_TON_Wait := FALSE;
                   #li_StepCase := 220;
               END_IF;

           220: // Position vertical NFC

               "gtyp_VGR".vertical_Axis.di_Target_Position := "gtyp_VGR".di_Pos_NFC_vertical;
               "gtyp_VGR".vertical_Axis.x_Start_Positioning := TRUE;
               //"gtyp_VGR".vertical_Axis.i_PWM := 500;

